IF (Mach_Control.Ca_b.Error[18] AND Sys_Control.btn.System_Rrestbtn) OR
    (CCD. CaRec.Finish.RectifyResult<>0 AND  CaCCDMark AND  Ca_AlarmTon[13].Q ) THEN
	   CaCCDMark :=FALSE;
	   Ca_AlarmTon[12].IN:=FALSE;
END_IF	

IF Mach_Control.U.DT_iMode=1 AND  rCaUse[4].Q THEN
 Par.stDT_date.Ca_sucker1_JS :=Par.stDT_date.Ca_sucker1_JS+1;
END_IF

IF( HMI_Hour>=7  AND HMI_Hour<9) OR (HMI_Hour>=19  AND HMI_Hour<21) THEN
      IF Par.stDT_date.Ca_sucker1_JS>=Par.stDT_date.Ca_sucker1Set THEN
	      Mach_Control.Ca_b.Error[43]:=TRUE;//负极送片搬运吸盘计数到达设定值
      END_IF
END_IF
IF Mach_Control.DT_b.Ca_sucker1_JSclear THEN
   Par.stDT_date.Ca_sucker1_JS:=0;
END_IF  

IF Mach_Control.U.DT_iMode=1 AND  rCaUse[5].Q THEN
 Par.stDT_date.Ca_sucker2_JS :=Par.stDT_date.Ca_sucker2_JS+1;
END_IF

IF( HMI_Hour>=7  AND HMI_Hour<9) OR (HMI_Hour>=19  AND HMI_Hour<21) THEN
      IF Par.stDT_date.Ca_sucker2_JS>=Par.stDT_date.Ca_sucker2Set THEN
	      Mach_Control.Ca_b.Error[44]:=TRUE;//负极叠台搬运吸盘计数到达设定值
      END_IF
END_IF
IF Mach_Control.DT_b.Ca_sucker2_JSclear THEN
   Par.stDT_date.Ca_sucker2_JS:=0;
END_IF  
IF Mach_Control.U.DT_iMode=1 AND  rCaUse[6].Q THEN
 Par.stDT_date.Ca_sucker3_JS :=Par.stDT_date.Ca_sucker3_JS+1;
END_IF

IF( HMI_Hour>=7  AND HMI_Hour<9) OR (HMI_Hour>=19  AND HMI_Hour<21) THEN
      IF Par.stDT_date.Ca_sucker3_JS>=Par.stDT_date.Ca_sucker3Set THEN
	      Mach_Control.Ca_b.Error[45]:=TRUE;//负极流水线搬运吸盘计数到达设定值
      END_IF
END_IF
IF Mach_Control.DT_b.Ca_sucker3_JSclear THEN
   Par.stDT_date.Ca_sucker3_JS:=0;
END_IF  
(*
IF Ca_CCDNG>=10 THEN
		Mach_Control.Ca_b.Error[12]:=TRUE;//负极NG收纳盒满料报警
END_IF

IF Mach_Control.Ca_b.Error[12] AND P2M2_sysControl.btn.System_Rrestbtn THEN
		 Mach_Control.Ca_b.Error[12]:=FALSE;
		 Ca_CCDNG:=0;
END_IF

*)
END_ACTION

ACTION Ca_Cahebelt:
Ca_TON[9].IN:=Mach_Control.Ca_b.bCa_PoleHave;
IF Ca_TON[9].Q THEN
	Mach_Control.Ca_b.bCa_PoleHave:=FALSE;//负极取流水线极片完成，
END_IF


//取料中信号复位
Ca_TON[10].IN:= NOT  arrAxisCtrl[AxiseNo.AxisName.CaCarryingUpDown1].Cmd.arrbRealPoint[1] AND Mach_Control.Ca_b.JumpPiceReady AND Mach_Control.Ca_b.Ca_MainBelting;
IF Ca_TON[10].Q THEN
	IF NOT  arrAxisCtrl[AxiseNo.AxisName.CaCarryingUpDown1].Cmd.arrbRealPoint[1] THEN		
		arrAxisCtrl[AxiseNo.AxisName.CaCarryingUpDown1].Cmd.iGoSetPos:=1;//负极送片搬运升降上升至初始高度	
	ELSE
		arrAxisCtrl[AxiseNo.AxisName.CaCarryingUpDown1].Cmd.iGoSetPos:=0;//负极送片搬运升降上升至初始高度	
	END_IF
END_IF
Ca_TON[11].IN:=arrAxisCtrl[AxiseNo.AxisName.CaCarryingUpDown1].Cmd.arrbRealPoint[1] AND Mach_Control.Ca_b.JumpPiceReady AND Mach_Control.Ca_b.Ca_MainBelting;
IF Ca_TON[11].Q  THEN
	Ca_StandbyStep2:=0;
	Mach_Control.Ca_b.Ca_BeltDone:=TRUE;//取流水线取极片完成
	Mach_Control.Ca_b.Ca_MainBelting:=FALSE;//正极搬运升降取极片中
END_IF




IF Mach_Control.U.DT_iMode=1 OR AG  THEN//在自动状态下
//负极模切分段皮带极片自动
CASE Ca_StandbyStep2  OF
0://判断取模切分板皮带机械手有无料标记
	IF NOT DP_SinStepe THEN
		IF   arrAxisCtrl[AxiseNo.AxisName.CaCarryingUpDown1].Status.Enabled  AND  arrAxisCtrl[AxiseNo.AxisName.CaCarryingLine1].Status.Enabled 
		AND  arrAxisCtrl[AxiseNo.AxisName.CaCarryingWhirling1].Status.Enabled  THEN
			IF Mach_Control.Ca_b.Ca_SegbeltFalg  THEN//负极取模切分段机械手有极片标记
				DT_SingeMode();//单步选择
				Ca_StandbyStep2:=100;
			ELSE//负极取模切分段机械手无料
				
				DT_SingeMode();//单步选择
				Ca_StandbyStep2:=10;
			END_IF
		END_IF
	END_IF
10://负极送片搬运升降轴上升至安全位，真空关闭
	IF NOT DP_SinStepe THEN
		arrCyCtrl[arrCyNo.ElectValveName.CaCarryingVacuum1]	.Cmd.bOFF:=TRUE;//负极搬运1真空关
		arrCyCtrl[arrCyNo.ElectValveName.CaCarryingVacuum1]	.Cmd.bON:=FALSE;//负极搬运1真空开
		IF arrAxisCtrl[AxiseNo.AxisName.CaCarryingUpDown1].Status.Homed AND arrAxisCtrl[AxiseNo.AxisName.CaCarryingUpDown1].Status.NoMoving AND 
			NOT arrAxisCtrl[AxiseNo.AxisName.CaCarryingUpDown1].Status.Error THEN
				IF arrAxisCtrl[AxiseNo.AxisName.CaCarryingUpDown1].Cmd.arrbRealPoint[1] THEN
					arrAxisCtrl[AxiseNo.AxisName.CaCarryingUpDown1].Cmd.iGoSetPos:=0;
					DT_SingeMode();//单步选择
					Ca_StandbyStep2:=20;
				ELSE
					arrAxisCtrl[AxiseNo.AxisName.CaCarryingUpDown1].Cmd.iGoSetPos:=1;//负极搬运升降1移动至初始高度
				END_IF
		END_IF
	END_IF
20://负极送片搬运平移至模切分段皮带取料位,负极搬运旋转1旋转至初始位
	IF NOT DP_SinStepe THEN
		IF arrAxisCtrl[AxiseNo.AxisName.CaCarryingUpDown1].Cmd.arrbRealPoint[1] AND  arrAxisCtrl[AxiseNo.AxisName.CaCarryingLine1].Status.Homed AND 
			arrAxisCtrl[AxiseNo.AxisName.CaCarryingLine1].Status.NoMoving AND NOT arrAxisCtrl[AxiseNo.AxisName.CaCarryingLine1].Status.Error THEN
			IF arrAxisCtrl[AxiseNo.AxisName.CaCarryingLine1].Cmd.arrbRealPoint[1] THEN
				arrAxisCtrl[AxiseNo.AxisName.CaCarryingLine1].Cmd.iGoSetPos:=0;
			ELSE
				arrAxisCtrl[AxiseNo.AxisName.CaCarryingLine1].Cmd.iGoSetPos:=1;//负极搬运升降1移动至初始高度
			END_IF
		END_IF
		IF arrAxisCtrl[AxiseNo.AxisName.CaCarryingUpDown1].Cmd.arrbRealPoint[1] AND  arrAxisCtrl[AxiseNo.AxisName.CaCarryingWhirling1].Status.Homed AND
			 arrAxisCtrl[AxiseNo.AxisName.CaCarryingWhirling1].Status.NoMoving AND NOT arrAxisCtrl[AxiseNo.AxisName.CaCarryingWhirling1].Status.Error THEN
			IF arrAxisCtrl[AxiseNo.AxisName.CaCarryingWhirling1].Cmd.arrbRealPoint[1] THEN
				arrAxisCtrl[AxiseNo.AxisName.CaCarryingWhirling1].Cmd.iGoSetPos:=0;
			ELSE
				arrAxisCtrl[AxiseNo.AxisName.CaCarryingWhirling1].Cmd.iGoSetPos:=1;//负极搬运旋转至初始位
			END_IF
		END_IF
		IF arrAxisCtrl[AxiseNo.AxisName.CaCarryingLine1].Cmd.arrbRealPoint[1]  AND arrAxisCtrl[AxiseNo.AxisName.CaCarryingWhirling1].Cmd.arrbRealPoint[1] THEN
			DT_SingeMode();//单步选择
			Ca_StandbyStep2:=30;
		END_IF
	END_IF

	

100://负极送片搬运升降轴上升至安全位，真空关闭
	IF NOT DP_SinStepe THEN
		IF arrAxisCtrl[AxiseNo.AxisName.CaCarryingUpDown1].Status.Homed AND arrAxisCtrl[AxiseNo.AxisName.CaCarryingUpDown1].Status.NoMoving AND 
			NOT arrAxisCtrl[AxiseNo.AxisName.CaCarryingUpDown1].Status.Error THEN
			IF arrAxisCtrl[AxiseNo.AxisName.CaCarryingUpDown1].Cmd.arrbRealPoint[1] THEN
						arrAxisCtrl[AxiseNo.AxisName.CaCarryingUpDown1].Cmd.iGoSetPos:=0;
						DT_SingeMode();//单步选择
						Ca_StandbyStep2:=110;
			ELSE
				arrAxisCtrl[AxiseNo.AxisName.CaCarryingUpDown1].Cmd.iGoSetPos:=1;//负极搬运升降1移动至初始高度
			END_IF
		END_IF
	END_IF
110://负极送片搬运平移至模切分段皮带放极片位, 负极搬运旋转1旋转至放位
	IF NOT DP_SinStepe THEN
		IF arrAxisCtrl[AxiseNo.AxisName.CaCarryingUpDown1].Cmd.arrbRealPoint[1] AND  arrAxisCtrl[AxiseNo.AxisName.CaCarryingLine1].Status.Homed AND 
			arrAxisCtrl[AxiseNo.AxisName.CaCarryingLine1].Status.NoMoving AND NOT arrAxisCtrl[AxiseNo.AxisName.CaCarryingLine1].Status.Error THEN
			IF arrAxisCtrl[AxiseNo.AxisName.CaCarryingLine1].Cmd.arrbRealPoint[2] THEN
				arrAxisCtrl[AxiseNo.AxisName.CaCarryingLine1].Cmd.iGoSetPos:=0;
			ELSE
				arrAxisCtrl[AxiseNo.AxisName.CaCarryingLine1].Cmd.iGoSetPos:=2;//负极搬运升降1移动至放极片位
			END_IF
		END_IF
		IF arrAxisCtrl[AxiseNo.AxisName.CaCarryingUpDown1].Cmd.arrbRealPoint[1] AND  arrAxisCtrl[AxiseNo.AxisName.CaCarryingWhirling1].Status.Homed AND
			 arrAxisCtrl[AxiseNo.AxisName.CaCarryingWhirling1].Status.NoMoving AND NOT arrAxisCtrl[AxiseNo.AxisName.CaCarryingWhirling1].Status.Error THEN
			IF arrAxisCtrl[AxiseNo.AxisName.CaCarryingWhirling1].Cmd.arrbRealPoint[2] THEN
				arrAxisCtrl[AxiseNo.AxisName.CaCarryingWhirling1].Cmd.iGoSetPos:=0;
			ELSE
				arrAxisCtrl[AxiseNo.AxisName.CaCarryingWhirling1].Cmd.iGoSetPos:=2;//负极搬运旋转至放极片位
			END_IF
		END_IF
		IF arrAxisCtrl[AxiseNo.AxisName.CaCarryingLine1].Cmd.arrbRealPoint[2]  AND arrAxisCtrl[AxiseNo.AxisName.CaCarryingWhirling1].Cmd.arrbRealPoint[2] THEN
			DT_SingeMode();//叠片单步选择
			Ca_StandbyStep2:=120;
		END_IF
	END_IF
120://判断负极流水线是否允许放极片  OR Mach_Control.U.EmptyRunMode
	IF NOT DP_SinStepe THEN
		IF Mach_Control.Ca_b.Ca_CacheBeltFLOK AND  Mach_Control.Ca_b.Ca_SegbeltFalg THEN
			DT_SingeMode();//单步选择
			Ca_StandbyStep2:=130;
		ELSIF NOT Mach_Control.Ca_b.Ca_SegbeltFalg THEN
			Ca_StandbyStep2:=0;
		END_IF
	END_IF
130://负极搬运升降1下降至放极片位
	IF NOT DP_SinStepe THEN
		IF arrAxisCtrl[AxiseNo.AxisName.CaCarryingLine1].Cmd.arrbRealPoint[2]  AND arrAxisCtrl[AxiseNo.AxisName.CaCarryingWhirling1].Cmd.arrbRealPoint[2] AND 
			arrAxisCtrl[AxiseNo.AxisName.CaCarryingUpDown1].Status.Homed AND arrAxisCtrl[AxiseNo.AxisName.CaCarryingUpDown1].Status.NoMoving AND 
			NOT arrAxisCtrl[AxiseNo.AxisName.CaCarryingUpDown1].Status.Error THEN
			IF arrAxisCtrl[AxiseNo.AxisName.CaCarryingUpDown1].Cmd.arrbRealPoint[3] THEN
				arrAxisCtrl[AxiseNo.AxisName.CaCarryingUpDown1].Cmd.iGoSetPos:=0;
				arrCyCtrl[arrCyNo.ElectValveName.CaCarryingVacuum1].Cmd.bOFF:=TRUE;//负极搬运1升降真空关
				arrCyCtrl[arrCyNo.ElectValveName.CaCarryingVacuum1].Cmd.bON:=FALSE;//负极搬运1升降真空关
				arrCyCtrl[arrCyNo.ElectValveName.CaCarryingVacuumBark1].Cmd.bON:=TRUE;//负极搬运1升降破真空开
				arrCyCtrl[arrCyNo.ElectValveName.CaCarryingVacuumBark1].Cmd.bOFF:=FALSE;//负极搬运1升降破真空开
				Mach_Control.Ca_b.Ca_SegbeltFalg:=FALSE;//置位负极取模切分段机械手有极片标记
				Par.stDT_date.Ca_betlCount.0:=TRUE;//置位负极片流水线放片位有片
				Par.stDT_date.Ca_MQ_Slice[1]:=Par.stDT_date.Ca_MQ_Slice[0];
				DT_SingeMode();//单步选择
				Ca_StandbyStep2:=140;
			ELSE
				arrAxisCtrl[AxiseNo.AxisName.CaCarryingUpDown1].Cmd.iGoSetPos:=3;//负极搬运升降1移动至放极片高度
			END_IF
		ELSE
			IF arrAxisCtrl[AxiseNo.AxisName.CaCarryingLine1].Cmd.arrbRealPoint[2] THEN
				arrAxisCtrl[AxiseNo.AxisName.CaCarryingLine1].Cmd.iGoSetPos:=0;
			ELSE
				arrAxisCtrl[AxiseNo.AxisName.CaCarryingLine1].Cmd.iGoSetPos:=2;//负极搬运升降1移动至放极片位
			END_IF	
			IF arrAxisCtrl[AxiseNo.AxisName.CaCarryingWhirling1].Cmd.arrbRealPoint[2] THEN
				arrAxisCtrl[AxiseNo.AxisName.CaCarryingWhirling1].Cmd.iGoSetPos:=0;
			ELSE
				arrAxisCtrl[AxiseNo.AxisName.CaCarryingWhirling1].Cmd.iGoSetPos:=2;//负极搬运旋转至放极片位
			END_IF			
		END_IF
	END_IF
140://负极送片搬运升降轴上升至安全位，真空关闭
	IF NOT DP_SinStepe THEN
		IF arrAxisCtrl[AxiseNo.AxisName.CaCarryingUpDown1].Status.Homed AND arrAxisCtrl[AxiseNo.AxisName.CaCarryingUpDown1].Status.NoMoving AND 
			NOT arrAxisCtrl[AxiseNo.AxisName.CaCarryingUpDown1].Status.Error THEN
			IF arrAxisCtrl[AxiseNo.AxisName.CaCarryingUpDown1].Cmd.arrbRealPoint[1] THEN
				arrAxisCtrl[AxiseNo.AxisName.CaCarryingUpDown1].Cmd.iGoSetPos:=0;
				DT_SingeMode();//单步选择
				Ca_StandbyStep2:=0;
			ELSE
				arrAxisCtrl[AxiseNo.AxisName.CaCarryingUpDown1].Cmd.iGoSetPos:=1;//负极搬运升降1移动至初始高度
			END_IF
		END_IF
	END_IF				
END_CASE	
END_IF


//负极缓存流水线缓存极片自动	
CASE Ca_StandbyStep4 OF
0://判断是否可以补极片,负极搬运升降1轴在安全位，负极搬运各项降2轴在安全位，负极流水线放极片端有极片，负极片流水线取级片端没极片 
	IF NOT Par.stDT_date.Ca_betlCount.5 AND Par.stDT_date.Ca_betlCount.0 AND  Mach_Control.Ca_b.Ca_betlMoveOK  THEN
		IF NOT Mach_Control.se.Offloadingsensor THEN
				Par.stDT_date.Ca_betlCount.4:=FALSE;
		END_IF
		Ca_StandbyStep4:=10;
	ELSIF	Ca_StandbyStep2=120 AND NOT Par.stDT_date.Ca_betlCount.5 AND Par.stDT_date.Ca_betlCount.0  AND  NOT  arrAxisCtrl[AxiseNo.AxisName.CaCarryingUpDown1].Cmd.arrbRealPoint[1] THEN
               // ( arrAxisCtrl[AxiseNo.AxisName.CaCarryingUpDown1].Status.fSetPos > arrAxisPar[AxiseNo.AxisName.CaCarryingUpDown1].arrTargetPoint[1]+0.5 OR
                //  arrAxisCtrl[AxiseNo.AxisName.CaCarryingUpDown1].Status.fSetPos < arrAxisPar[AxiseNo.AxisName.CaCarryingUpDown1].arrTargetPoint[1]-0.5)THEN
		         Mach_Control.Ca_b.Error[41]:=TRUE;//负极缓存皮带准备运动时，负极升降1不在安全位报警	
	END_IF
10://负极流水线皮带向前移动固定距离
	arrAxisCtrl[AxiseNo.AxisName.CaBelt].Cmd.bDynamitcsParSel:=1;	
	arrAxisPar[AxiseNo.AxisName.CaBelt].fTagatTime:=Par.stDT_date.BeltPoistTime;
	arrAxisCtrl[AxiseNo.AxisName.CaBelt].Cmd.fPosition_of_Rel:=Par.stDT_date.BeltPoistSet;
	arrAxisCtrl[AxiseNo.AxisName.CaBelt].Cmd.bMoveRel:=TRUE;	
	Ca_StandbyStep4:=20;
20:
	IF NOT arrAxisCtrl[AxiseNo.AxisName.CaBelt].Cmd.bMoveRel THEN
		Par.stDT_date.Ca_betlCount:=SHL(Par.stDT_date.Ca_betlCount,1);//极片向前移一位
		Ca_StandbyStep4:=31;
	END_IF

31:	
	Par.stDT_date.Ca_MQ_Slice[6]:=Par.stDT_date.Ca_MQ_Slice[5];
	Ca_StandbyStep4:=32;

32:
	Par.stDT_date.Ca_MQ_Slice[5]:=Par.stDT_date.Ca_MQ_Slice[4];
	Ca_StandbyStep4:=33;

33:
	Par.stDT_date.Ca_MQ_Slice[4]:=Par.stDT_date.Ca_MQ_Slice[3];
	Ca_StandbyStep4:=34;

34:	
	Par.stDT_date.Ca_MQ_Slice[3]:=Par.stDT_date.Ca_MQ_Slice[2];
	Ca_StandbyStep4:=35;

35:
	Par.stDT_date.Ca_MQ_Slice[2]:=Par.stDT_date.Ca_MQ_Slice[1];
	Ca_StandbyStep4:=36;

36://复位负极片流水线放片位有片
	MEMSET(ADR(Par.stDT_date.Ca_MQ_Slice[1]),0,SIZEOF(Par.stDT_date.Ca_MQ_Slice[1]));
	Par.stDT_date.Ca_betlCount.0:=FALSE;
	Ca_StandbyStep4:=0;
END_CASE


CASE Ca_StandbyStep2  OF
30://判断模切分段皮带是否允许取极片 OR Mach_Control.U.EmptyRunMode 
	IF NOT DP_SinStepe THEN
		IF Mach_Control.Ca_b.Ca_MainBeltOK THEN
			Mach_Control.Ca_b.Ca_MainBelting:=TRUE;//负极模切分段皮带取极片中
			arrCyCtrl[arrCyNo.ElectValveName.CaCarryingVacuum1]	.Cmd.bON:=TRUE;//负极搬运1真空打开
			arrCyCtrl[arrCyNo.ElectValveName.CaCarryingVacuum1]	.Cmd.bOFF:=FALSE;//负极搬运1真空关闭
			DT_SingeMode();//单步选择
			Ca_StandbyStep2:=35;
		//ELSE
		//	Ca_StandbyStep2:=0;
		END_IF
	END_IF
35://负极搬动升降1下降取极片
	IF NOT DP_SinStepe THEN
		IF arrAxisCtrl[AxiseNo.AxisName.CaCarryingLine1].Cmd.arrbRealPoint[1]  AND arrAxisCtrl[AxiseNo.AxisName.CaCarryingWhirling1].Cmd.arrbRealPoint[1] AND 
			arrAxisCtrl[AxiseNo.AxisName.CaCarryingUpDown1].Status.Homed AND  NOT arrAxisCtrl[AxiseNo.AxisName.CaCarryingUpDown1].Status.Error THEN
			IF arrAxisCtrl[AxiseNo.AxisName.CaCarryingUpDown1].Cmd.arrbRealPoint[2] OR arrAxisCtrl[AxiseNo.AxisName.CaCarryingUpDown1].Status.Moving THEN
				arrAxisCtrl[AxiseNo.AxisName.CaCarryingUpDown1].Cmd.iGoSetPos:=0;
				DT_SingeMode();//单步选择
				Ca_TON[6].IN:=FALSE;
				Ca_StandbyStep2:=40;
			ELSE
				arrAxisCtrl[AxiseNo.AxisName.CaCarryingUpDown1].Cmd.iGoSetPos:=2;//负极搬运升降1移动至初始高度
			END_IF					
		END_IF
	END_IF
40://负极搬动升降1下降取极片
	IF arrAxisCtrl[AxiseNo.AxisName.CaCarryingLine1].Cmd.arrbRealPoint[1]  AND arrAxisCtrl[AxiseNo.AxisName.CaCarryingWhirling1].Cmd.arrbRealPoint[1] AND 
	arrAxisCtrl[AxiseNo.AxisName.CaCarryingUpDown1].Status.Homed AND arrAxisCtrl[AxiseNo.AxisName.CaCarryingUpDown1].Status.NoMoving AND 
	NOT arrAxisCtrl[AxiseNo.AxisName.CaCarryingUpDown1].Status.Error THEN
		IF arrAxisCtrl[AxiseNo.AxisName.CaCarryingUpDown1].Cmd.arrbRealPoint[2] THEN			
			IF NOT Ca_TON[6].Q THEN
				Ca_TON[6].IN:=TRUE;
			ELSE
				//Mach_Control.Ca_b.bCa_PoleHave:=TRUE;//负极取流水线极片完成，复位取片位置极片有无信号
				arrAxisCtrl[AxiseNo.AxisName.CaCarryingUpDown1].Cmd.iGoSetPos:=0;
				//arrCyCtrl[arrCyNo.ElectValveName.CaMQBeltVacuum].Cmd.bOFF:=TRUE;//负极模切分段皮带真空关闭
				//arrCyCtrl[arrCyNo.ElectValveName.CaMQBeltVacuum].Cmd.bON:=FALSE;//负极模切分段皮带真空关闭
				//arrCyCtrl[arrCyNo.ElectValveName.CaMQBeltVacuumBark].Cmd.bON:=TRUE;//负极模切分段皮带破真空打开
				Mach_Control.Ca_b.Ca_SegbeltFalg:=TRUE;//置位负极取模切分段机械手有极片标记
				Par.stDT_date.Ca_MQ_Slice[0]:=Par.stDT_date.CaMQ_MES;//转移皮带上的数据
				DT_SingeMode();//单步选择
				Ca_TON[6].IN:=FALSE;
				Ca_StandbyStep2:=50;								
			END_IF								
		ELSE
			arrAxisCtrl[AxiseNo.AxisName.CaCarryingUpDown1].Cmd.iGoSetPos:=2;//负极搬运升降1移动至初始高度
		END_IF					
	END_IF

50://
	//20240414 wcz
    IF   arrAxisCtrl[AxiseNo.AxisName.CaCarryingUpDown1].Status.fActPos<=(arrAxisPar[AxiseNo.AxisName.CaCarryingUpDown1].arrTargetPoint[2]-3) AND
		 arrAxisCtrl[AxiseNo.AxisName.CaCarryingUpDown1].Status.Moving THEN
			Mach_Control.Ca_b.Ca_MainBelting:=FALSE;//负极模切分段皮带取极片中
			Mach_Control.Ca_b.Ca_BeltDone:=TRUE;//负极取主流水线极片完成		 
			Mach_Control.Ca_b.bCa_PoleHave:=TRUE;//负极取流水线极片完成，复位取片位置极片有无信号
	END_IF

	IF arrAxisCtrl[AxiseNo.AxisName.CaCarryingUpDown1].Status.Homed AND arrAxisCtrl[AxiseNo.AxisName.CaCarryingUpDown1].Status.NoMoving AND 
	NOT arrAxisCtrl[AxiseNo.AxisName.CaCarryingUpDown1].Status.Error THEN
		IF arrAxisCtrl[AxiseNo.AxisName.CaCarryingUpDown1].Cmd.arrbRealPoint[1] THEN
			arrAxisCtrl[AxiseNo.AxisName.CaCarryingUpDown1].Cmd.iGoSetPos:=0;
			Mach_Control.Ca_b.Ca_MainBelting:=FALSE;//负极模切分段皮带取极片中
			Mach_Control.Ca_b.Ca_BeltDone:=TRUE;//负极取主流水线极片完成
			DT_SingeMode();//单步选择
			Ca_StandbyStep2:=0;
		ELSE
			arrAxisCtrl[AxiseNo.AxisName.CaCarryingUpDown1].Cmd.iGoSetPos:=1;//负极搬运升降1移动至初始高度
		END_IF
	END_IF
END_CASE
END_ACTION

ACTION Ca_Cam:
Ca_Cam_ton[1](PT:=T#100MS);
Ca_Cam_ton[2](PT:=T#100MS);
Ca_Cam_ton[3](PT:=T#100MS);
Ca_Cam_ton[4](PT:=T#100MS);
Ca_Cam_ton[5](PT:=T#100MS);
(***********************************负极凸轮表创建************************************************)
(*
      fbCaCrectCamCarryingLine1              :FB_CrectCamMove ;
      fbCaCrectCamCarryingUpDown1       :FB_CrectCamUpDown ;
      fbCaCrectCamCarryingLine2             :FB_CrectCamMove ;
      fbCaCrectCamCarryingUpDown2       :FB_CrectCamUpDown ;
      fbCaCrectCamDTCarryingLine            :FB_CrectCamMove ;
      fbCaCrectCamDTCarryingUpDown     :FB_CrectCamUpDown ;
*)
//负极取流水线搬运平移凸轮创建
fbCaCrectCamCarryingLine1(
	bCreatTable:=                fbCaCrectCamCarryingLine1.bCreatTable , 
	Reset:=                          stSysState.bReset  ,  
	iTable:=                       TableNo.M_CaCarryingLine1  , 
	fMoveLength:=             390 , 
	fMasterKeyPos:=          224 , 
	
	axisMaster:=                 arrAxis[AxiseNo.VirAxisName.CaCarryingVirGM] ,  
    axisSlave:=                    arrAxis[AxiseNo.AxisName.CaCarryingLine1] ,  
	bCreatTableDone=> , 
	bCreatTableError=> , 
	bError=> );

fbCaCrectCamCarryingLine1.bCreatTableDone;
fbCaCrectCamCarryingLine1.bCreatTableError;
fbCaCrectCamCarryingLine1.bError;

//负极取流水线搬运放片升降凸轮创建
fbCaCrectCamCarryingUpDown1(
	bCreatTable:=                         fbCaCrectCamCarryingUpDown1.bCreatTable , 
	Reset:=                                  stSysState.bReset  ,  
	iTable:=                                   TableNo.M_CaCarryingUpDown1   , 
	fMoveLength:=                        18   , //升降轴放片或取片位
	fSaveLength:=                          3, //升降轴安全位
	fInitLength:=						      13,//升降轴耦合初始位
	fMasterKeyPos1:= , //208
	fMasterKeyPos2:= , //256
	fMasterKeyPos3:= , //328

    axisMaster:=                        arrAxis[AxiseNo.VirAxisName.CaCarryingVirGM] ,   
	axisSlave:=                           arrAxis[AxiseNo.AxisName.CaCarryingUpDown1] ,  

	bCreatTableDone=> , 
	bCreatTableError=> , 
	bError=> );
fbCaCrectCamCarryingUpDown1.bCreatTableDone;
fbCaCrectCamCarryingUpDown1.bCreatTableError;
fbCaCrectCamCarryingUpDown1.bError;

//负极取流水线搬运取片升降凸轮创建
fbCaCrectCamCarryingUpDown1_1(
	bCreatTable:=                         fbCaCrectCamCarryingUpDown1_1.bCreatTable , 
	Reset:=                                  stSysState.bReset  ,  
	iTable:=                                   TableNo.M_CaCarryingUpDown1_1   , 
	fMoveLength:=                        18   , //升降轴放片或取片位
	fSaveLength:=                          3, //升降轴安全位
	fInitLength:=						      13,//升降轴耦合初始位
	fMasterKeyPos1:= , //208
	fMasterKeyPos2:= , //256
	fMasterKeyPos3:= , //328

    axisMaster:=                        arrAxis[AxiseNo.VirAxisName.CaCarryingVirGM] ,   
	axisSlave:=                           arrAxis[AxiseNo.AxisName.CaCarryingUpDown1] ,  

	bCreatTableDone=> , 
	bCreatTableError=> , 
	bError=> );
fbCaCrectCamCarryingUpDown1_1.bCreatTableDone;
fbCaCrectCamCarryingUpDown1_1.bCreatTableError;
fbCaCrectCamCarryingUpDown1_1.bError;

//负极取流水线旋转凸轮创建 
fbCaCrectCamCarryingWhirling(
	bCreatTable:=                fbCaCrectCamCarryingWhirling.bCreatTable , 
	Reset:=                          stSysState.bReset  ,  
	iTable:=                       TableNo.M_CaCarryingWhirling1  , 
	fMoveLength:=             390 , 
	fMasterKeyPos:=          170 , //224
	
	axisMaster:=                 arrAxis[AxiseNo.VirAxisName.CaCarryingVirGM] ,  
    axisSlave:=                    arrAxis[AxiseNo.AxisName.CaCarryingWhirling1] ,  
	bCreatTableDone=> , 
	bCreatTableError=> , 
	bError=> );

fbCaCrectCamCarryingWhirling.bCreatTableDone;
fbCaCrectCamCarryingWhirling.bCreatTableError;
fbCaCrectCamCarryingWhirling.bError;




//负极送纠偏平台搬运平移凸轮创建
fbCaCrectCamCarryingLine2.fMoveLength:=ABS(arrAxisPar[AxiseNo.AxisName.CaCarryingLine2].arrTargetPoint[1]-arrAxisPar[AxiseNo.AxisName.CaCarryingLine2].arrTargetPoint[2]);
fbCaCrectCamCarryingLine2(
	bCreatTable:=                fbCaCrectCamCarryingLine2.bCreatTable , 
	Reset:=                          stSysState.bReset  ,  
	iTable:=                       TableNo.M_CaCarryingLine2  , 
	fMoveLength:=             , 
	fMasterKeyPos:=          250 , //
	
	axisMaster:=                 arrAxis[AxiseNo.VirAxisName.VirMain] ,  
    axisSlave:=                    arrAxis[AxiseNo.AxisName.CaCarryingLine2] ,  
	bCreatTableDone=> , 
	bCreatTableError=> , 
	bError=> );

fbCaCrectCamCarryingLine2.bCreatTableDone;
fbCaCrectCamCarryingLine2.bCreatTableError;
fbCaCrectCamCarryingLine2.bError;


(**********20240528SJ***************)
arrAxisPar[AxiseNo.AxisName.CaCarryingUpDown2].arrTargetPoint[10]:=10; //等待高度  参数可调
arrAxisPar[AxiseNo.AxisName.CaCarryingUpDown2].arrTargetPoint[11]:=25; //安全高度  参数可调
arrAxisPar[AxiseNo.AxisName.CaCarryingUpDown2].arrTargetPoint[4]:=arrAxisPar[AxiseNo.AxisName.CaCarryingUpDown2].arrTargetPoint[3]-arrAxisPar[AxiseNo.AxisName.CaCarryingUpDown2].arrTargetPoint[10];  //等待位置
//arrAxisPar[AxiseNo.AxisName.AnCarryingUpDown].arrTargetPoint[1]:=arrAxisPar[AxiseNo.AxisName.AnCarryingUpDown].arrTargetPoint[3]-arrAxisPar[AxiseNo.AxisName.AnCarryingUpDown].arrTargetPoint[11];  //安全位置

//负极送纠偏平台搬运升降取片凸轮创建 20240509 CF
fbCaCrectCamCarryingUpDown2(  //取片
	bCreatTable:=                         fbCaCrectCamCarryingUpDown2.bCreatTable , 
	Reset:=                                  stSysState.bReset  ,  
	iTable:=                                   TableNo.M_CaCarryingUpDown2   , 
	fMoveLength:=4, //取片高度
	fSaveLength:=arrAxisPar[AxiseNo.AxisName.CaCarryingUpDown2].arrTargetPoint[10] - arrAxisPar[AxiseNo.AxisName.CaCarryingUpDown2].arrTargetPoint[11],//安全高度
	//fInitLength:=arrAxisPar[AxiseNo.AxisName.CaCarryingUpDown2].arrTargetPoint[4],//升降轴耦合初始位
	fMasterKeyPos1:=110 , //
	fMasterKeyPos2:=250 , //144
	//fMasterKeyPos3:=240 , //198
	//fMasterKeyPos4:=310 , //324
	
    axisMaster:=                        arrAxis[AxiseNo.VirAxisName.VirMain] ,   
	axisSlave:=                           arrAxis[AxiseNo.AxisName.CaCarryingUpDown2] ,  

	bCreatTableDone=> , 
	bCreatTableError=> , 
	bError=> );
fbCaCrectCamCarryingUpDown2.bCreatTableDone;
fbCaCrectCamCarryingUpDown2.bCreatTableError;
fbCaCrectCamCarryingUpDown2.bError;


//负极送纠偏平台搬运升降放极片凸轮创建-
fbCaCrectCamCarryingUpDown2_1(   //--------放片
	bCreatTable:=                         fbCaCrectCamCarryingUpDown2_1.bCreatTable , 
	Reset:=                                  stSysState.bReset  ,  
	iTable:=                                   TableNo.M_CaCarryingUpDown2_1   , 
	fMoveLength:= arrAxisPar[AxiseNo.AxisName.CaCarryingUpDown2].arrTargetPoint[10]       ,//放片高度
	fSaveLength:=arrAxisPar[AxiseNo.AxisName.CaCarryingUpDown2].arrTargetPoint[10] - arrAxisPar[AxiseNo.AxisName.CaCarryingUpDown2].arrTargetPoint[11]  , //安全高度
	//fInitLength:=arrAxisPar[AxiseNo.AxisName.CaCarryingUpDown2].arrTargetPoint[4],//升降轴耦合初始位
	fMasterKeyPos1:=110 , //125
	fMasterKeyPos2:=250 , //
	fMasterKeyPos3:=260 , //
	fMasterKeyPos4:=320 , //
	fMasterKeyPos5:=359 , //
	//fMasterKeyPos6:=250 , //
	fSlaveVelo:=0.25 , //
	
    axisMaster:=                        arrAxis[AxiseNo.VirAxisName.VirMain] ,   
	axisSlave:=                           arrAxis[AxiseNo.AxisName.CaCarryingUpDown2] ,  

	bCreatTableDone=> , 
	bCreatTableError=> , 
	bError=> );
fbCaCrectCamCarryingUpDown2_1.bCreatTableDone;
fbCaCrectCamCarryingUpDown2_1.bCreatTableError;
fbCaCrectCamCarryingUpDown2_1.bError;

//负极送纠偏平台搬运升降放极片凸轮创建-
fbCaCrectCamCarryingUpDown2_3(   //--------放片
	bCreatTable:=                         fbCaCrectCamCarryingUpDown2_3.bCreatTable , 
	Reset:=                                   stSysState.bReset  ,  
	iTable:=                                  TableNo.M_CaCarryingUpDown2_3   , 
	//fMoveLength:= arrAxisPar[AxiseNo.AxisName.CaCarryingUpDown2].arrTargetPoint[10]       ,//放片高度
	fSaveLength:=arrAxisPar[AxiseNo.AxisName.CaCarryingUpDown2].arrTargetPoint[10] - arrAxisPar[AxiseNo.AxisName.CaCarryingUpDown2].arrTargetPoint[11]  , //安全高度
	//fInitLength:=arrAxisPar[AxiseNo.AxisName.CaCarryingUpDown2].arrTargetPoint[4],//升降轴耦合初始位
	fMasterKeyPos1:=110 , //130
	fMasterKeyPos2:=250 , //
	//fMasterKeyPos3:=260 , //
	//fMasterKeyPos4:=320 , //
	//fMasterKeyPos5:=359 , //
	//fMasterKeyPos6:=250 , //
	//fSlaveVelo:=0.25 , //
	
    axisMaster:=                        arrAxis[AxiseNo.VirAxisName.VirMain] ,   
	axisSlave:=                           arrAxis[AxiseNo.AxisName.CaCarryingUpDown2] ,  

	bCreatTableDone=> , 
	bCreatTableError=> , 
	bError=> );
fbCaCrectCamCarryingUpDown2_3.bCreatTableDone;
fbCaCrectCamCarryingUpDown2_3.bCreatTableError;
fbCaCrectCamCarryingUpDown2_3.bError;




//负极叠片搬运平移凸轮创建
fbCaCrectCamDTCarryingLine.fMoveLength:=ABS(arrAxisPar[AxiseNo.AxisName.CaDTCarryingLine].arrTargetPoint[1]- arrAxisPar[AxiseNo.AxisName.CaDTCarryingLine].arrTargetPoint[2]);
fbCaCrectCamDTCarryingLine(
	bCreatTable:=                fbCaCrectCamDTCarryingLine.bCreatTable , 
	Reset:=                          stSysState.bReset  ,  
	iTable:=                        TableNo.M_CaDTCarryingLine  , 
	fMoveLength:=              , 
	fMasterKeyPos:=          250 , //
	
	axisMaster:=                 arrAxis[AxiseNo.VirAxisName.VirMain] ,  
    axisSlave:=                    arrAxis[AxiseNo.AxisName.CaDTCarryingLine] ,  
	bCreatTableDone=> , 
	bCreatTableError=> , 
	bError=> );

fbCaCrectCamDTCarryingLine.bCreatTableDone;
fbCaCrectCamDTCarryingLine.bCreatTableError;
fbCaCrectCamDTCarryingLine.bError;



(**********20240528SJ***************)
arrAxisPar[AxiseNo.AxisName.CaDTCarryingUpDown].arrTargetPoint[10]:=6; //等待高度  参数可调
arrAxisPar[AxiseNo.AxisName.CaDTCarryingUpDown].arrTargetPoint[11]:=18; //抬升高度  参数可调
arrAxisPar[AxiseNo.AxisName.CaDTCarryingUpDown].arrTargetPoint[4]:=arrAxisPar[AxiseNo.AxisName.CaDTCarryingUpDown].arrTargetPoint[3]-arrAxisPar[AxiseNo.AxisName.CaDTCarryingUpDown].arrTargetPoint[10];  //等待位置    以放片位为基准
//arrAxisPar[AxiseNo.AxisName.AnDTCarryingUpDown].arrTargetPoint[1]:=arrAxisPar[AxiseNo.AxisName.AnDTCarryingUpDown].arrTargetPoint[3]-arrAxisPar[AxiseNo.AxisName.AnDTCarryingUpDown].arrTargetPoint[11];  //安全位置

//负极叠片搬运升降取片凸轮创建
fbCaCrectCamDTCarryingUpDown(//取片
	bCreatTable:=                         fbCaCrectCamDTCarryingUpDown.bCreatTable , 
	Reset:=                                  stSysState.bReset  ,  
	iTable:=                                   TableNo.M_CaDTCarryingUpDown   , 
	fMoveLength:=arrAxisPar[AxiseNo.AxisName.CaDTCarryingUpDown].arrTargetPoint[10]-(arrAxisPar[AxiseNo.AxisName.CaDTCarryingUpDown].arrTargetPoint[3]-arrAxisPar[AxiseNo.AxisName.CaDTCarryingUpDown].arrTargetPoint[2])               ,//取片高度
	fSaveLength:=arrAxisPar[AxiseNo.AxisName.CaDTCarryingUpDown].arrTargetPoint[10]-arrAxisPar[AxiseNo.AxisName.CaDTCarryingUpDown].arrTargetPoint[11]              , //安全位
	//fInitLength:=arrAxisPar[AxiseNo.AxisName.CaDTCarryingUpDown].arrTargetPoint[4],//升降轴耦合初始位
	fMasterKeyPos1:=125 , //
	fMasterKeyPos2:=250 , //
	fMasterKeyPos3:=260 , //
	fMasterKeyPos4:= 320, //
	fMasterKeyPos5:=359 , //
	fMasterKeyPos6:= , //
	fSlaveVelo:=0.25 , //
	
    axisMaster:=                        arrAxis[AxiseNo.VirAxisName.VirMain] ,   
	axisSlave:=                           arrAxis[AxiseNo.AxisName.CaDTCarryingUpDown] ,  

	bCreatTableDone=> , 
	bCreatTableError=> , 
	bError=> );
fbCaCrectCamDTCarryingUpDown.bCreatTableDone;
fbCaCrectCamDTCarryingUpDown.bCreatTableError;
fbCaCrectCamDTCarryingUpDown.bError;


//负极叠片搬运升降放片凸轮创建
IF  DP_Step0>3000 AND DP_Step0<=3080 THEN
     fbCaCrectCamDTCarryingUpDown1.iTableSel:=2;
ELSE	 
	 fbCaCrectCamDTCarryingUpDown1.iTableSel:=1;
END_IF		 

fbCaCrectCamDTCarryingUpDown1(//放片
	bCreatTable:=                         fbCaCrectCamDTCarryingUpDown1.bCreatTable , 
	Reset:=                                   stSysState.bReset  ,  
	iTable:=                                   TableNo.M_CaDTCarryingUpDown1   , 
	bCamIn:=  fbCaCamInDTCarryingUpDown.bCamInExecute AND  fbCaCamInDTCarryingUpDown.iTableSel=2    , 
	fMoveLength:=arrAxisPar[AxiseNo.AxisName.CaDTCarryingUpDown].arrTargetPoint[10] , //取片高度
	fSaveLength:=arrAxisPar[AxiseNo.AxisName.CaDTCarryingUpDown].arrTargetPoint[10]-arrAxisPar[AxiseNo.AxisName.CaDTCarryingUpDown].arrTargetPoint[11]  , //安全高度
	//fInitLength:=arrAxisPar[AxiseNo.AxisName.CaDTCarryingUpDown].arrTargetPoint[4] ,//升降轴耦合初始位
	fMasterKeyPos1:=120 , //208
	fMasterKeyPos2:=250 , //256
	fMasterKeyPos3:=260 , //256
	fMasterKeyPos4:=342 , //328
	fMasterKeyPos5:=359 , //328
	fSlaveVelo:=0.25 , //
    axisMaster:=                        arrAxis[AxiseNo.VirAxisName.VirMain] ,   
	axisSlave:=                           arrAxis[AxiseNo.AxisName.CaDTCarryingUpDown] ,  

	bCreatTableDone=> , 
	bCreatTableError=> , 
	bError=> );
fbCaCrectCamDTCarryingUpDown1.bCreatTableDone;
fbCaCrectCamDTCarryingUpDown1.bCreatTableError;
fbCaCrectCamDTCarryingUpDown1.bError;


//正极叠片搬运升降避让凸轮创建
fbCaCrectCamDTCarryingUpDown3(//放片
	bCreatTable:=fbCaCrectCamDTCarryingUpDown3.bCreatTable, 
	Reset:=stSysState.bReset  , 
	iTable:=TableNo.M_CaDTCarryingUpDown3 , 
	//fMoveLength:=arrAxisPar[AxiseNo.AxisName.AnDTCarryingUpDown].arrTargetPoint[10] ,//放片高度 
	fSaveLength:=arrAxisPar[AxiseNo.AxisName.CaDTCarryingUpDown].arrTargetPoint[10]-arrAxisPar[AxiseNo.AxisName.CaDTCarryingUpDown].arrTargetPoint[11]  , //安全高度
	//fInitLength:=arrAxisPar[AxiseNo.AxisName.AnDTCarryingUpDown].arrTargetPoint[4],//升降轴耦合初始位
	fMasterKeyPos1:=130 , //208
	fMasterKeyPos2:=260 , //256
	//fMasterKeyPos3:=260 , //256
	//fMasterKeyPos4:=342 , //328
//	fMasterKeyPos5:=359 , //328
//	fSlaveVelo:=0.25 , //
	axisSlave:=arrAxis[AxiseNo.AxisName.CaDTCarryingUpDown]  , 
	axisMaster:=arrAxis[AxiseNo.VirAxisName.VirMain]  , 
	bCreatTableDone=> , 
	bCreatTableError=> , 
	bError=> );
	
fbCaCrectCamDTCarryingUpDown3.bCreatTableDone;
fbCaCrectCamDTCarryingUpDown3.bCreatTableError;
fbCaCrectCamDTCarryingUpDown3.bError;











tCaCreate_TON(IN:= , PT:=T#0.5S , Q=> , ET=> );
IF Mach_Control.U.DT_iMode=3 OR Mach_Control.U.DT_iMode=0 THEN//在手动状态下
				//在触摸屏上生成凸轮
				//rCaCreate_TRIG(CLK:=Mach_Control.Ca_b.CreateCamStart , Q=> );	
				rCaCreate_TRIG(CLK:=(Mach_Control.Ca_b.CreateCamStart 
                                    AND	NOT arrAxisCtrl[AxiseNo.AxisName.CaCarryingLine2].Status.Coupled
									AND	NOT arrAxisCtrl[AxiseNo.AxisName.CaCarryingUpDown2].Status.Coupled
									AND	NOT arrAxisCtrl[AxiseNo.AxisName.CaDTCarryingLine].Status.Coupled
									AND	NOT arrAxisCtrl[AxiseNo.AxisName.CaDTCarryingUpDown].Status.Coupled), Q=> );				
				IF rCaCreate_TRIG.Q THEN
					tCaCreate_TON.IN:=FALSE;
					CaCrectCamStep0:=10;
					Mach_Control.Ca_b.Error[0]:=FALSE;
				END_IF
END_IF
				//负极取料凸轮自动创建
				CASE CaCrectCamStep0 OF
						10:
								IF NOT tCaCreate_TON.Q THEN
										//fbCaCrectCamCarryingLine1.bCreatTable :=TRUE;//负极取流水线平移凸轮创建
										//fbCaCrectCamCarryingUpDown1.bCreatTable:=TRUE;//负极取流水线放片升降凸轮创建
										//fbCaCrectCamCarryingUpDown1_1.bCreatTable:=TRUE;//负极取流水线取片升降凸轮创建
										//fbCaCrectCamCarryingWhirling.bCreatTable:=TRUE;//负极取流水线旋转凸轮创建
										 fbCaCrectCamCarryingLine2.bCreatTable :=FALSE;//负极送片搬运平移凸轮创建
										 fbCaCrectCamCarryingUpDown2.bCreatTable:=FALSE;//负极送片搬运升降取片凸轮创建
										 fbCaCrectCamCarryingUpDown2_1.bCreatTable:=FALSE;//负极送片搬运升降放片凸轮创建
										 fbCaCrectCamCarryingUpDown2_3.bCreatTable:=FALSE;//负极送片搬运升降放片凸轮创建
										 fbCaCrectCamDTCarryingLine.bCreatTable :=FALSE;//负极叠片搬运平移凸轮创建
										 fbCaCrectCamDTCarryingUpDown.bCreatTable:=FALSE;//负极叠片搬运升降取片凸轮创建
										 fbCaCrectCamDTCarryingUpDown1.bCreatTable:=FALSE;//负极叠片搬运升降放片凸轮创建
										  fbCaCrectCamDTCarryingUpDown3.bCreatTable:=FALSE;//负极叠片搬运升降放片凸轮创建
										 Mach_Control.Ca_b.CreateCamDone:=FALSE;
										 tCaCreate_TON.IN:=TRUE;					
								ELSE
											tCaCreate_TON.IN:=FALSE;	
											CaCrectCamStep0:=11;
								END_IF
								
						11:	
								IF  NOT Ca_Cam_ton[1].Q THEN
									arrAxisCtrl[AxiseNo.AxisName.CaCarryingLine2].Cmd.bStop:=TRUE;
									arrAxisCtrl[AxiseNo.AxisName.CaCarryingUpDown2].Cmd.bStop:=TRUE;
									arrAxisCtrl[AxiseNo.AxisName.CaDTCarryingLine].Cmd.bStop:=TRUE;
									arrAxisCtrl[AxiseNo.AxisName.CaDTCarryingUpDown].Cmd.bStop:=TRUE;
									Ca_Cam_ton[1].IN:=TRUE;
								ELSE
									Ca_Cam_ton[1].IN:=FALSE;
									CaCrectCamStep0:=12;
									arrAxisCtrl[AxiseNo.AxisName.CaCarryingLine2].Cmd.bStop:=FALSE;
									arrAxisCtrl[AxiseNo.AxisName.CaCarryingUpDown2].Cmd.bStop:=FALSE;
									arrAxisCtrl[AxiseNo.AxisName.CaDTCarryingLine].Cmd.bStop:=FALSE;
									arrAxisCtrl[AxiseNo.AxisName.CaDTCarryingUpDown].Cmd.bStop:=FALSE;
								END_IF
								
						12:
								IF  NOT Ca_Cam_ton[2].Q THEN
									arrAxisCtrl[AxiseNo.AxisName.CaCarryingLine2].Cmd.bReset:=TRUE;	
									arrAxisCtrl[AxiseNo.AxisName.CaCarryingUpDown2].Cmd.bReset:=TRUE;
									arrAxisCtrl[AxiseNo.AxisName.CaDTCarryingLine].Cmd.bReset:=TRUE;
									arrAxisCtrl[AxiseNo.AxisName.CaDTCarryingUpDown].Cmd.bReset:=TRUE;
									Ca_Cam_ton[2].IN:=TRUE;
								 ELSE
									 Ca_Cam_ton[2].IN:=FALSE;
									 CaCrectCamStep0:=13;
									arrAxisCtrl[AxiseNo.AxisName.CaCarryingLine2].Cmd.bReset:=FALSE;	
									arrAxisCtrl[AxiseNo.AxisName.CaCarryingUpDown2].Cmd.bReset:=FALSE;
									arrAxisCtrl[AxiseNo.AxisName.CaDTCarryingLine].Cmd.bReset:=FALSE;
									arrAxisCtrl[AxiseNo.AxisName.CaDTCarryingUpDown].Cmd.bReset:=FALSE;
								 END_IF
							

						13:
							arrAxisCtrl[AxiseNo.AxisName.CaCarryingLine2].Cmd.bEnable:=TRUE;
							arrAxisCtrl[AxiseNo.AxisName.CaCarryingUpDown2].Cmd.bEnable:=TRUE;
							arrAxisCtrl[AxiseNo.AxisName.CaDTCarryingLine].Cmd.bEnable:=TRUE;
							arrAxisCtrl[AxiseNo.AxisName.CaDTCarryingUpDown].Cmd.bEnable:=TRUE;
							IF arrAxisCtrl[AxiseNo.AxisName.CaCarryingLine2].Status.Enabled AND arrAxisCtrl[AxiseNo.AxisName.CaCarryingUpDown2].Status.Enabled AND
								arrAxisCtrl[AxiseNo.AxisName.CaDTCarryingLine].Status.Enabled AND arrAxisCtrl[AxiseNo.AxisName.CaDTCarryingUpDown].Status.Enabled THEN
								 CaCrectCamStep0:=20;
							END_IF
								
								
						20://凸轮创建
									//fbCaCrectCamCarryingLine1.bCreatTable :=TRUE;//负极取流水线平移凸轮创建
									//fbCaCrectCamCarryingUpDown1.bCreatTable:=TRUE;//负极取流水线放片升降凸轮创建
									//fbCaCrectCamCarryingUpDown1_1.bCreatTable:=TRUE;//负极取流水线取片升降凸轮创建
									//fbCaCrectCamCarryingWhirling.bCreatTable:=TRUE;//负极取流水线旋转凸轮创建
									 fbCaCrectCamCarryingLine2.bCreatTable :=TRUE;//负极送片搬运平移凸轮创建
									 fbCaCrectCamCarryingUpDown2.bCreatTable:=TRUE;//负极送片搬运升降取片凸轮创建
									 fbCaCrectCamCarryingUpDown2_1.bCreatTable:=TRUE;//负极送片搬运升降放片凸轮创建
									 fbCaCrectCamCarryingUpDown2_3.bCreatTable:=TRUE;//负极送片搬运升降放片凸轮创建
									 fbCaCrectCamDTCarryingLine.bCreatTable :=TRUE;//负极叠片搬运平移凸轮创建
									 fbCaCrectCamDTCarryingUpDown.bCreatTable:=TRUE;//负极叠片搬运升降取片凸轮创建
									 fbCaCrectCamDTCarryingUpDown1.bCreatTable:=TRUE;//负极叠片搬运升降放片凸轮创建
									  fbCaCrectCamDTCarryingUpDown3.bCreatTable:=TRUE;//负极叠片搬运升降放片凸轮创建
									 Mach_Control.Ca_b.CreateCamDone:=FALSE;
									 CaCrectCamStep0:=30;
						30://判断凸轮是否创建完成
									IF fbCaCrectCamCarryingLine2.bCreatTableDone AND  fbCaCrectCamCarryingUpDown2.bCreatTableDone AND  fbCaCrectCamCarryingUpDown2_1.bCreatTableDone  AND
										 fbCaCrectCamDTCarryingLine.bCreatTableDone AND fbCaCrectCamDTCarryingUpDown.bCreatTableDone AND fbCaCrectCamDTCarryingUpDown1.bCreatTableDone  AND
                                        fbCaCrectCamCarryingUpDown2_3.bCreatTableDone AND  fbCaCrectCamDTCarryingUpDown3.bCreatTableDone  THEN
											Mach_Control.Ca_b.CreateCamDone:=TRUE;
											CaCrectCamStep0:=6666;
									ELSE
											IF fbCaCrectCamCarryingLine2.bCreatTableError OR fbCaCrectCamCarryingUpDown2.bCreatTableError OR fbCaCrectCamCarryingUpDown2_1.bCreatTableError  OR 
												fbCaCrectCamDTCarryingLine.bCreatTableError OR fbCaCrectCamDTCarryingUpDown.bCreatTableError OR  fbCaCrectCamDTCarryingUpDown1.bCreatTableError OR 
                                          fbCaCrectCamCarryingUpDown2_3.bCreatTableError OR  fbCaCrectCamDTCarryingUpDown3.bCreatTableError    THEN								
												Mach_Control.Ca_b.Error[0]:=TRUE;//负极取片创建凸轮报警
												CaCrectCamStep0:=9999;
											END_IF
									END_IF
				END_CASE




(***********************************负极凸轮耦合***********************************************)
(*
      fbCaCamInCarryingLine1                      :FB_CamIn ;    
      fbCaCamInCarryingUpDown1               :FB_CamIn ;    
      fbCaCamInCarryingLine2                     :FB_CamIn ;    
      fbCaCamInCarryingUpDown2              :FB_CamIn ;    
      fbCaCamInDTCarryingLine                   :FB_CamIn ;    
      fbCaCamInDTCarryingUpDown            :FB_CamIn ;    
*)

//负极取流水线搬运平移凸轮耦合
fbCaCamInCarryingLine1.ParCamIn.SlaveScaling;
fbCaCamInCarryingLine1(
	Reset:=                      stSysState.bReset  , 
	bCamInExecute:=       fbCaCamInCarryingLine1.bCamInExecute, 
	iTable1:=                   TableNo.M_CaCarryingLine1  , 
	iTable2:=                   , 
	iTableSel:=                 , 
	ParCamIn:= , 
  	axisMaster:=            arrAxis[AxiseNo.VirAxisName.CaCarryingVirGM] ,  
	axisSlave:=               arrAxis[AxiseNo.AxisName.CaCarryingLine1] ,  
	bError=> , 
	bReady=> , 
	bInSync=> );

(*Mach_Control.Ca_b.Error[11]:=*)fbCaCamInCarryingLine1.bError;
fbCaCamInCarryingLine1.bReady;
fbCaCamInCarryingLine1.bInSync;

//负极取流水线搬运升降凸轮耦合
fbCaCamInCarryingUpDown1.iTableSel;
fbCaCamInCarryingUpDown1(
	Reset:=                      stSysState.bReset  , 
	bCamInExecute:=       fbCaCamInCarryingUpDown1.bCamInExecute, 
	iTable1:=                   TableNo.M_CaCarryingUpDown1  , 
	iTable2:=                   TableNo.M_CaCarryingUpDown1_1 , 
	iTableSel:=                  , 
	ParCamIn:=                  , 
  	axisMaster:=            arrAxis[AxiseNo.VirAxisName.CaCarryingVirGM] ,  
	axisSlave:=               arrAxis[AxiseNo.AxisName.CaCarryingUpDown1] ,  
	bError=> , 
	bReady=> , 
	bInSync=> );

(*Mach_Control.Ca_b.Error[12]:=*)fbCaCamInCarryingUpDown1.bError;
fbCaCamInCarryingUpDown1.bReady;
fbCaCamInCarryingUpDown1.bInSync;
//负极取流水线旋转
fbCaCamInCarryingWhirling.ParCamIn.SlaveScaling;
fbCaCamInCarryingWhirling(
	Reset:=                      stSysState.bReset  , 
	bCamInExecute:=       fbCaCamInCarryingWhirling.bCamInExecute, 
	iTable1:=                   TableNo.M_CaCarryingWhirling1  , 
	iTable2:=                   , 
	iTableSel:=                 , 
	ParCamIn:= , 
  	axisMaster:=            arrAxis[AxiseNo.VirAxisName.CaCarryingVirGM] ,  
	axisSlave:=               arrAxis[AxiseNo.AxisName.CaCarryingWhirling1] ,  
	bError=> , 
	bReady=> , 
	bInSync=> );

fbCaCamInCarryingWhirling.bError;
fbCaCamInCarryingWhirling.bReady;
fbCaCamInCarryingWhirling.bInSync;




//负极送片搬运平移凸轮耦合
fbCaCamInCarryingLine2.ParCamIn.SlaveScaling;
fbCaCamInCarryingLine2.ParCamIn.MasterScaling:=fCaScaling;//20240508 CF
fbCaCamInCarryingLine2(
	Reset:=                      stSysState.bReset  , 
	bCamInExecute:=       fbCaCamInCarryingLine2.bCamInExecute, 
	iTable1:=                   TableNo.M_CaCarryingLine2  , 
	iTable2:=                   , 
	iTableSel:=                 , 
	ParCamIn:= , 
  	axisMaster:=            arrAxis[AxiseNo.VirAxisName.VirMain] ,  
	axisSlave:=               arrAxis[AxiseNo.AxisName.CaCarryingLine2] ,  
	bError=> , 
	bReady=> , 
	bInSync=> );
(*Mach_Control.Ca_b.Error[13]:=*)fbCaCamInCarryingLine2.bError;
fbCaCamInCarryingLine2.bReady;
fbCaCamInCarryingLine2.bInSync;


//负极送纠偏搬动升降凸轮耦合
fbCaCamInCarryingUpDown2.ParCamIn.MasterScaling:=fCaScaling;//20240508 CF
fbCaCamInCarryingUpDown2(
	Reset:=                      stSysState.bReset  , 
	bCamInExecute:=       fbCaCamInCarryingUpDown2.bCamInExecute, 
	iTable1:=                   TableNo.M_CaCarryingUpDown2  , 
	iTable2:=                   TableNo.M_CaCarryingUpDown2_1  , 
	iTable3:=                   TableNo.M_CaCarryingUpDown2_3  , 
	iTableSel:=                  , //耦合凸轮选择
	ParCamIn:=                  , 
  	axisMaster:=            arrAxis[AxiseNo.VirAxisName.VirMain] ,  
	axisSlave:=               arrAxis[AxiseNo.AxisName.CaCarryingUpDown2] ,  
	bError=> , 
	bReady=> , 
	bInSync=> );

(*Mach_Control.Ca_b.Error[14]:=*)fbCaCamInCarryingUpDown2.bError;
fbCaCamInCarryingUpDown2.bReady;
fbCaCamInCarryingUpDown2.bInSync;


//负极叠台搬运平移凸轮耦合
fbCaCamInDTCarryingLine.ParCamIn.SlaveScaling;
fbCaCamInDTCarryingLine(
	Reset:=                      stSysState.bReset  , 
	bCamInExecute:=       fbCaCamInDTCarryingLine.bCamInExecute, 
	iTable1:=                   TableNo.M_CaDTCarryingLine  , 
	iTable2:=                   , 
	iTableSel:=                 , 
	ParCamIn:=                , 
  	axisMaster:=            arrAxis[AxiseNo.VirAxisName.VirMain] ,  
	axisSlave:=               arrAxis[AxiseNo.AxisName.CaDTCarryingLine] ,  
	bError=> , 
	bReady=> , 
	bInSync=> );
(*Mach_Control.Ca_b.Error[15]:=*)fbCaCamInDTCarryingLine.bError;
fbCaCamInDTCarryingLine.bReady;
fbCaCamInDTCarryingLine.bInSync;


//负极叠台搬运升降凸轮耦合
fbCaCamInDTCarryingUpDown(
	Reset:=                      stSysState.bReset  , 
	bCamInExecute:=       fbCaCamInDTCarryingUpDown.bCamInExecute, 
	iTable1:=                   TableNo.M_CaDTCarryingUpDown  , 
	iTable2:=                    TableNo.M_CaDTCarryingUpDown1, 
	iTable3:=                    TableNo.M_CaDTCarryingUpDown3, 
	iTableSel:=                  , 
	ParCamIn:=                  , 
  	axisMaster:=            arrAxis[AxiseNo.VirAxisName.VirMain] ,  
	axisSlave:=               arrAxis[AxiseNo.AxisName.CaDTCarryingUpDown] ,  
	bError=> , 
	bReady=> , 
	bInSync=> );

(*Mach_Control.Ca_b.Error[16]:=*)fbCaCamInDTCarryingUpDown.bError;
fbCaCamInDTCarryingUpDown.bReady;
fbCaCamInDTCarryingUpDown.bInSync;


IF fbCaCamInCarryingLine1.bError OR fbCaCamInCarryingUpDown1.bError OR fbCaCamInCarryingLine2.bError OR fbCaCamInCarryingUpDown2.bError OR fbCaCamInDTCarryingLine.bError OR fbCaCamInDTCarryingUpDown.bError THEN
		Mach_Control.Ca_b.Error[11]:=TRUE;//负极藕合凸轮报警
	ELSE	
		Mach_Control.Ca_b.Error[11]:=FALSE;
END_IF
END_ACTION

ACTION Ca_Conditions:
(********************负极放弃取片********************)
Mach_Control.Ca_b.JumpPiceReady:=Mach_Control.U.DT_iMode<>1 OR Mach_Control.Ca_b.Ca_SegbeltFalg OR Mach_Control.U.EmptyRunMode OR   (Mach_Control.DT_b.SinStepMode AND Ca_StandbyStep2<>35 AND Ca_StandbyStep2<>40);

(********************负极取片准备好********************)
Mach_Control.Ca_b.GetPiceReady:=NOT Mach_Control.Ca_b.JumpPiceReady AND
														arrAxisCtrl[AxiseNo.AxisName.CaCarryingUpDown1].Status.Homed AND arrAxisCtrl[AxiseNo.AxisName.CaCarryingUpDown1].Cmd.arrbRealPoint[1] AND
														arrAxisCtrl[AxiseNo.AxisName.CaCarryingLine1].Status.Homed AND arrAxisCtrl[AxiseNo.AxisName.CaCarryingLine1].Cmd.arrbRealPoint[1];
(*
IF Mach_Control.U.DT_iMode=1 AND NOT Mach_Control.Ca_b.Ca_SegbeltFalg AND (DP_Step0<>6030 AND DP_Step0<>6040 AND 
Mach_Control.An_b.An_Quantited <= Par.stDT_date.An_Quantity  AND  Mach_Control.Ca_b.Ca_Quantited < Par.stDT_date.Ca_Quantity) AND
   arrAxisCtrl[AxiseNo.AxisName.CaCarryingUpDown1].Status.Homed AND arrAxisCtrl[AxiseNo.AxisName.CaCarryingUpDown1].Cmd.arrbRealPoint[1] AND
   arrAxisCtrl[AxiseNo.AxisName.CaCarryingLine1].Status.Homed AND arrAxisCtrl[AxiseNo.AxisName.CaCarryingLine1].Cmd.arrbRealPoint[1] THEN
 		Mach_Control.Ca_b.GetPiceReady:=TRUE;
ELSE
 		Mach_Control.Ca_b.GetPiceReady:=FALSE;	
END_IF

IF Mach_Control.U.DT_iMode<>1 OR Mach_Control.Ca_b.Ca_SegbeltFalg OR JumpPiceReady_temp1 OR JumpPiceReady_temp2 OR JumpPiceReady_temp3 THEN
	Mach_Control.Ca_b.JumpPiceReady:=TRUE;
ELSE
	Mach_Control.Ca_b.JumpPiceReady:=FALSE;
END_IF
*)



//负极纠偏平台放极片允许
IF  NOT Mach_Control.Ca_b.Ca_deviationFalg AND arrAxisCtrl[AxiseNo.AxisName.CadeviationX1].Status.Homed AND NOT arrAxisCtrl[AxiseNo.AxisName.CadeviationX1].Status.Error AND 
	arrAxisCtrl[AxiseNo.AxisName.CadeviationX1].Status.NoMoving AND arrAxisCtrl[AxiseNo.AxisName.CadeviationX1].Cmd.arrbRealPoint[1] AND 
	arrAxisCtrl[AxiseNo.AxisName.CadeviationX2].Status.Homed AND NOT arrAxisCtrl[AxiseNo.AxisName.CadeviationX2].Status.Error AND 
	arrAxisCtrl[AxiseNo.AxisName.CadeviationX2].Status.NoMoving AND arrAxisCtrl[AxiseNo.AxisName.CadeviationX2].Cmd.arrbRealPoint[1] AND 
	arrAxisCtrl[AxiseNo.AxisName.CadeviationY].Status.Homed AND NOT arrAxisCtrl[AxiseNo.AxisName.CadeviationY].Status.Error AND 
	arrAxisCtrl[AxiseNo.AxisName.CadeviationY].Status.NoMoving AND arrAxisCtrl[AxiseNo.AxisName.CadeviationY].Cmd.arrbRealPoint[1] THEN
	Mach_Control.Ca_b.Ca_deviationFPOK:=TRUE;
ELSE
	Mach_Control.Ca_b.Ca_deviationFPOK:=FALSE;	
END_IF

//负极搬运皮带取极片允许
IF  Par.stDT_date.Ca_betlCount.5 AND arrAxisCtrl[AxiseNo.AxisName.CaBelt].Status.NoMoving AND NOT arrAxisCtrl[AxiseNo.AxisName.CaBelt].Status.Error THEN
	Mach_Control.Ca_b.Ca_CacheBeltDLOK:=TRUE;
ELSE
	Mach_Control.Ca_b.Ca_CacheBeltDLOK:=FALSE;	
END_IF



//负极搬运皮带放极片允许
IF NOT  Par.stDT_date.Ca_betlCount.0 AND arrAxisCtrl[AxiseNo.AxisName.CaCarryingUpDown1].Status.NoMoving AND NOT arrAxisCtrl[AxiseNo.AxisName.CaCarryingUpDown1].Status.Error  THEN
	Mach_Control.Ca_b.Ca_CacheBeltFLOK:=TRUE;
ELSE
	Mach_Control.Ca_b.Ca_CacheBeltFLOK:=FALSE;
END_IF
//负极搬运升降1、负极搬运升降2允许负极流水线电机转动   根据实际情况修改 20240509 CF
IF ((arrAxisCtrl[AxiseNo.AxisName.CaCarryingUpDown1].Status.fSetPos <= arrAxisPar[AxiseNo.AxisName.CaCarryingUpDown1].arrTargetPoint[3]-4
	  AND arrAxisCtrl[AxiseNo.AxisName.CaCarryingUpDown1].Status.Homed ) OR
	 (arrAxisCtrl[AxiseNo.AxisName.CaCarryingLine1].Status.fActPos < arrAxisPar[AxiseNo.AxisName.CaCarryingLine1].arrTargetPoint[2]-100  
	  AND arrAxisCtrl[AxiseNo.AxisName.CaCarryingLine1].Status.Homed ) ) AND
	 
	 ((arrAxisCtrl[AxiseNo.AxisName.CaCarryingUpDown2].Status.fSetPos <= arrAxisPar[AxiseNo.AxisName.CaCarryingUpDown2].arrTargetPoint[2]-4
	   AND arrAxisCtrl[AxiseNo.AxisName.CaCarryingUpDown2].Status.Homed ) OR 
	   (arrAxisCtrl[AxiseNo.AxisName.CaCarryingLine2].Status.fActPos > arrAxisPar[AxiseNo.AxisName.CaCarryingLine2].arrTargetPoint[1]+225  
	     AND  arrAxisCtrl[AxiseNo.AxisName.CaCarryingLine2].Status.Homed ) ) THEN
	Mach_Control.Ca_b.Ca_betlMoveOK:=TRUE;
ELSE
	Mach_Control.Ca_b.Ca_betlMoveOK:=FALSE;	
END_IF


(*  南昌备份
IF ((arrAxisCtrl[AxiseNo.AxisName.CaCarryingUpDown1].Status.fSetPos <= arrAxisPar[AxiseNo.AxisName.CaCarryingUpDown1].arrTargetPoint[1]+0.5)
	 OR arrAxisCtrl[AxiseNo.AxisName.CaCarryingLine1].Cmd.arrbRealPoint[1]) AND arrAxisCtrl[AxiseNo.AxisName.CaCarryingUpDown1].Status.Homed AND
	 
	 ((arrAxisCtrl[AxiseNo.AxisName.CaCarryingUpDown2].Status.fSetPos <= arrAxisPar[AxiseNo.AxisName.CaCarryingUpDown2].arrTargetPoint[4]+0.5) 
	OR arrAxisCtrl[AxiseNo.AxisName.CaCarryingLine2].Cmd.arrbRealPoint[2]) AND arrAxisCtrl[AxiseNo.AxisName.CaCarryingUpDown1].Status.Homed  THEN
	Mach_Control.Ca_b.Ca_betlMoveOK:=TRUE;
ELSE
	Mach_Control.Ca_b.Ca_betlMoveOK:=FALSE;	
END_IF
*)


//负极搬运平移2在安全位,、负极叠片升降在安全位、尾卷夹隔膜平移在安全位、允许负极叠片搬运平移移动纠偏平台位
//arrAxisCtrl[AxiseNo.AxisName.TailCurlSEPTALine].Status.Homed  AND arrAxisCtrl[AxiseNo.AxisName.TailCurlSEPTALine].Status.fActPos <= arrAxisPar[AxiseNo.AxisName.TailCurlSEPTALine].arrTargetPoint[1] 
IF arrAxisCtrl[AxiseNo.AxisName.CaCarryingLine2].Status.Homed AND arrAxisCtrl[AxiseNo.AxisName.CaCarryingLine2].Status.NoMoving AND arrAxisCtrl[AxiseNo.AxisName.CaCarryingLine2].Cmd.arrbRealPoint[1] AND
    arrAxisCtrl[AxiseNo.AxisName.CaDTCarryingUpDown].Status.Homed AND arrAxisCtrl[AxiseNo.AxisName.CaDTCarryingUpDown].Status.NoMoving AND  TailCurlSEPTA_SafePos AND
 	 arrAxisCtrl[AxiseNo.AxisName.CaDTCarryingUpDown].Status.fSetPos   <=arrAxisPar[AxiseNo.AxisName.CaDTCarryingUpDown].arrTargetPoint[4]+0.1 THEN
	Mach_Control.Ca_b.CarryingSafepos[0]:=TRUE;
ELSE
	Mach_Control.Ca_b.CarryingSafepos[0]:=FALSE;	
END_IF
//隔膜平移在正极片位、负极叠片搬运升降在安全位，允许负极叠片搬运平移至叠片位
IF arrAxisCtrl[AxiseNo.AxisName.SEPTATLine].Status.Homed  AND arrAxisCtrl[AxiseNo.AxisName.SEPTATLine].Status.NoMoving AND arrAxisCtrl[AxiseNo.AxisName.SEPTATLine].Cmd.arrbRealPoint[1] AND 
    arrAxisCtrl[AxiseNo.AxisName.CaDTCarryingUpDown].Status.Homed AND  arrAxisCtrl[AxiseNo.AxisName.CaDTCarryingUpDown].Status.NoMoving AND arrAxisCtrl[AxiseNo.AxisName.CaDTCarryingUpDown].Cmd.arrbRealPoint[1] AND
	arrAxis[AxiseNo.AxisName.TailCurlSEPTALine].Status.Homed  AND arrAxisCtrl[AxiseNo.AxisName.TailCurlSEPTALine].Status.fSetPos <= arrAxisPar[AxiseNo.AxisName.TailCurlSEPTALine].arrTargetPoint[1]   THEN
	Mach_Control.Ca_b.CarryingSafepos[1]:=TRUE;
ELSE
	Mach_Control.Ca_b.CarryingSafepos[1]:=FALSE;
END_IF
//负极送片搬运升降2在安全位，允许负极送片搬运2平移至取流水线极片位
IF arrAxisCtrl[AxiseNo.AxisName.CaCarryingUpDown2].Cmd.arrbRealPoint[1] AND arrAxisCtrl[AxiseNo.AxisName.CaCarryingLine2].Status.Homed AND
	arrAxisCtrl[AxiseNo.AxisName.CaCarryingLine2].Status.NoMoving THEN
	Mach_Control.Ca_b.CarryingSafepos[2]:=TRUE;
ELSE
	Mach_Control.Ca_b.CarryingSafepos[2]:=FALSE;
END_IF
//负极送片搬运升降2在安全位、负极叠片搬运在安全位，允许负极送片搬运2平移至纠偏位
IF arrAxisCtrl[AxiseNo.AxisName.CaCarryingUpDown2].Cmd.arrbRealPoint[1] AND arrAxisCtrl[AxiseNo.AxisName.CaCarryingUpDown2].Status.Homed AND
	arrAxisCtrl[AxiseNo.AxisName.CaCarryingUpDown2].Status.NoMoving AND arrAxisCtrl[AxiseNo.AxisName.CaDTCarryingLine].Status.Homed  AND 
	arrAxisCtrl[AxiseNo.AxisName.CaDTCarryingLine].Status.NoMoving AND arrAxisCtrl[AxiseNo.AxisName.CaDTCarryingLine].Cmd.arrbRealPoint[2]  THEN
	Mach_Control.Ca_b.CarryingSafepos[3]:=TRUE;
ELSE
	Mach_Control.Ca_b.CarryingSafepos[3]:=FALSE;
END_IF	
//负极送片搬运升降1在安全位，允许负极搬运平移1移动
IF  arrAxisCtrl[AxiseNo.AxisName.CaCarryingUpDown1].Cmd.arrbRealPoint[1] AND arrAxisCtrl[AxiseNo.AxisName.CaCarryingUpDown1].Status.Homed AND
	arrAxisCtrl[AxiseNo.AxisName.CaCarryingUpDown1].Status.NoMoving THEN
	Mach_Control.Ca_b.CarryingSafepos[4]:=TRUE;
ELSE
	Mach_Control.Ca_b.CarryingSafepos[4]:=FALSE;
END_IF		 
//负极送片搬运安全位，负极叠片搬运安全位，尾卷夹隔膜平移，允许纠偏平台移动
IF arrAxisCtrl[AxiseNo.AxisName.CaCarryingUpDown2].Status.Homed AND arrAxisCtrl[AxiseNo.AxisName.CaCarryingLine2].Status.Homed  AND 
	(arrAxisCtrl[AxiseNo.AxisName.CaCarryingUpDown2].Status.fSetPos<=(arrAxisPar[AxiseNo.AxisName.CaCarryingUpDown2].arrTargetPoint[4]+2) OR arrAxisCtrl[AxiseNo.AxisName.CaCarryingLine2].Cmd.arrbRealPoint[1]) AND 
    arrAxisCtrl[AxiseNo.AxisName.CaDTCarryingUpDown].Status.Homed AND arrAxisCtrl[AxiseNo.AxisName.CaDTCarryingLine].Status.Homed  AND 
	(arrAxisCtrl[AxiseNo.AxisName.CaDTCarryingUpDown].Status.fSetPos<=(arrAxisPar[AxiseNo.AxisName.CaDTCarryingUpDown].arrTargetPoint[4]+2) OR arrAxisCtrl[AxiseNo.AxisName.CaDTCarryingLine].Cmd.arrbRealPoint[2]) (*AND 
	arrAxisCtrl[AxiseNo.AxisName.TailCurlSEPTALine].Status.Homed AND arrAxisCtrl[AxiseNo.AxisName.TailCurlSEPTALine].Status.fActPos<=arrAxisPar[AxiseNo.AxisName.TailCurlSEPTALine].arrTargetPoint[1]  *) THEN
	Mach_Control.Ca_b.CarryingSafepos[5]:=TRUE;
ELSE
	Mach_Control.Ca_b.CarryingSafepos[5]:=FALSE;
END_IF		
//负极取流水线机械手在安全位，允许模切流水线移动
(*
IF arrAxisCtrl[AxiseNo.AxisName.CaCarryingUpDown1].Status.Homed AND NOT Mach_Control.Ca_b.Ca_MainBelting AND 
 	(arrAxisCtrl[AxiseNo.AxisName.CaCarryingUpDown1].Status.fSetPos<=arrAxisPar[AxiseNo.AxisName.CaCarryingUpDown1].arrTargetPoint[1]+0.2 OR 
	  arrAxisCtrl[AxiseNo.AxisName.CaCarryingLine1].Cmd.arrbRealPoint[1]	) THEN
	Mach_Control.Ca_b.Ca_BeltSafe:=TRUE;
ELSE
	Mach_Control.Ca_b.Ca_BeltSafe:=FALSE;
END_IF
*)
(*
IF  Mach_Control.Ca_b.Ca_MainBelting THEN
	Mach_Control.Ca_b.Ca_BeltSafe:=TRUE;
ELSIF NOT Mach_Control.Ca_b.Ca_MainBelting AND  arrAxisCtrl[AxiseNo.AxisName.CaCarryingUpDown1].Cmd.arrbRealPoint[4] THEN
	Mach_Control.Ca_b.Ca_BeltSafe:=FALSE;
END_IF
*)
IF  Mach_Control.Ca_b.Ca_MainBelting THEN
	Mach_Control.Ca_b.Ca_BeltSafe:=TRUE;
ELSE
	Mach_Control.Ca_b.Ca_BeltSafe:=FALSE;
END_IF
//负极主流水线取片完成延时复位
Ca_BeltTon(IN:=Mach_Control.Ca_b.Ca_BeltDone , PT:=T#20MS , Q=> , ET=> );
IF Ca_BeltTon.Q THEN
	Mach_Control.Ca_b.Ca_BeltDone:=FALSE;//复位主流水线取片完成
END_IF




/////////////////////////////////////////////////////////////
/////////////////////////////////////////////////////////
////////////////////////////////////////////电机条件

//负极送片皮带
IF Mach_Control.U.DT_iMode=3  AND arrAxisCtrl[AxiseNo.AxisName.CaCarryingUpDown1].Status.fActPos<= arrAxisPar[AxiseNo.AxisName.CaCarryingUpDown1].arrTargetPoint[1] +0.5
AND  arrAxisCtrl[AxiseNo.AxisName.CaCarryingUpDown2].Status.fActPos<=arrAxisPar[AxiseNo.AxisName.CaCarryingUpDown2].arrTargetPoint[4]+0.5  THEN
	arrAxisCtrl[AxiseNo.AxisName.CaBelt].Cmd.Home_Condition:=TRUE;
	arrAxisCtrl[AxiseNo.AxisName.CaBelt].Cmd.JogN_Condition:=TRUE;
	arrAxisCtrl[AxiseNo.AxisName.CaBelt].Cmd.JogP_Condition:=TRUE;
ELSE
	arrAxisCtrl[AxiseNo.AxisName.CaBelt].Cmd.Home_Condition:=FALSE;	
	arrAxisCtrl[AxiseNo.AxisName.CaBelt].Cmd.JogN_Condition:=FALSE;
	arrAxisCtrl[AxiseNo.AxisName.CaBelt].Cmd.JogP_Condition:=FALSE;
END_IF



//负极送片搬运1平移
IF Mach_Control.U.DT_iMode=3 AND arrAxisCtrl[AxiseNo.AxisName.CaCarryingUpDown1].Status.Homed AND
 	arrAxisCtrl[AxiseNo.AxisName.CaCarryingUpDown1].Status.fSetPos<= arrAxisPar[AxiseNo.AxisName.CaCarryingUpDown1].arrTargetPoint[1]+1 THEN
	arrAxisCtrl[AxiseNo.AxisName.CaCarryingLine1].Cmd.Home_Condition:=TRUE;
ELSE
arrAxisCtrl[AxiseNo.AxisName.CaCarryingLine1].Cmd.Home_Condition:=FALSE;	
END_IF

IF Mach_Control.U.DT_iMode=3 AND arrAxisCtrl[AxiseNo.AxisName.CaCarryingLine1].Status.Homed AND 
	arrAxisCtrl[AxiseNo.AxisName.CaCarryingUpDown1].Status.Homed AND
 	arrAxisCtrl[AxiseNo.AxisName.CaCarryingUpDown1].Status.fSetPos<= arrAxisPar[AxiseNo.AxisName.CaCarryingUpDown1].arrTargetPoint[1]+1 THEN
	arrAxisCtrl[AxiseNo.AxisName.CaCarryingLine1].Cmd.GoPoint_Condition[1]:=TRUE;
ELSE
	arrAxisCtrl[AxiseNo.AxisName.CaCarryingLine1].Cmd.GoPoint_Condition[1]:=FALSE;	
END_IF

IF Mach_Control.U.DT_iMode=3 AND arrAxisCtrl[AxiseNo.AxisName.CaCarryingLine1].Status.Homed AND
	arrAxisCtrl[AxiseNo.AxisName.CaCarryingUpDown1].Status.Homed AND
 	arrAxisCtrl[AxiseNo.AxisName.CaCarryingUpDown1].Status.fSetPos<= arrAxisPar[AxiseNo.AxisName.CaCarryingUpDown1].arrTargetPoint[1]+1 THEN
		arrAxisCtrl[AxiseNo.AxisName.CaCarryingLine1].Cmd.GoPoint_Condition[2]:=TRUE;
ELSE
		arrAxisCtrl[AxiseNo.AxisName.CaCarryingLine1].Cmd.GoPoint_Condition[2]:=FALSE;	
END_IF

//负极送片搬运1升降
IF Mach_Control.U.DT_iMode=3  THEN
	arrAxisCtrl[AxiseNo.AxisName.CaCarryingUpDown1].Cmd.Home_Condition:=TRUE;
ELSE
	arrAxisCtrl[AxiseNo.AxisName.CaCarryingUpDown1].Cmd.Home_Condition:=FALSE;	
END_IF

IF Mach_Control.U.DT_iMode=3 AND arrAxisCtrl[AxiseNo.AxisName.CaCarryingUpDown1].Status.Homed THEN
	arrAxisCtrl[AxiseNo.AxisName.CaCarryingUpDown1].Cmd.GoPoint_Condition[1]:=TRUE;
ELSE
	arrAxisCtrl[AxiseNo.AxisName.CaCarryingUpDown1].Cmd.GoPoint_Condition[1]:=FALSE;	
END_IF

IF arrAxisCtrl[AxiseNo.AxisName.CaCarryingLine1].Cmd.arrbRealPoint[1] AND  Mach_Control.U.DT_iMode=3 AND arrAxisCtrl[AxiseNo.AxisName.CaCarryingUpDown1].Status.Homed THEN
	arrAxisCtrl[AxiseNo.AxisName.CaCarryingUpDown1].Cmd.GoPoint_Condition[2]:=TRUE;
ELSE
	arrAxisCtrl[AxiseNo.AxisName.CaCarryingUpDown1].Cmd.GoPoint_Condition[2]:=FALSE;	
END_IF

IF arrAxisCtrl[AxiseNo.AxisName.CaCarryingLine1].Cmd.arrbRealPoint[2] AND  Mach_Control.U.DT_iMode=3 AND arrAxisCtrl[AxiseNo.AxisName.CaCarryingUpDown1].Status.Homed THEN
	arrAxisCtrl[AxiseNo.AxisName.CaCarryingUpDown1].Cmd.GoPoint_Condition[3]:=TRUE;
ELSE
	arrAxisCtrl[AxiseNo.AxisName.CaCarryingUpDown1].Cmd.GoPoint_Condition[3]:=FALSE;	
END_IF

//负极送片搬运2平移
IF Mach_Control.U.DT_iMode=3 AND arrAxisCtrl[AxiseNo.AxisName.CaCarryingUpDown2].Status.Homed AND
 arrAxisCtrl[AxiseNo.AxisName.CaCarryingUpDown2].Status.fSetPos<=arrAxisPar[AxiseNo.AxisName.CaCarryingUpDown2].arrTargetPoint[1]+1    AND
 arrCyCtrl[arrCyNo.CylinderName.CaScrapbinUDCy].Io.DIOFFSwitch  AND	 arrCyCtrl[arrCyNo.CylinderName.CaScrapbinCy].Io.DIOnSwitch  THEN
		arrAxisCtrl[AxiseNo.AxisName.CaCarryingLine2].Cmd.Home_Condition:=TRUE;
ELSE
		arrAxisCtrl[AxiseNo.AxisName.CaCarryingLine2].Cmd.Home_Condition:=FALSE;	
END_IF

IF Mach_Control.U.DT_iMode=3 AND arrAxisCtrl[AxiseNo.AxisName.CaCarryingUpDown2].Status.Homed AND
arrAxisCtrl[AxiseNo.AxisName.CaCarryingUpDown2].Status.fSetPos<=arrAxisPar[AxiseNo.AxisName.CaCarryingUpDown2].arrTargetPoint[1]+1 AND
 arrAxisCtrl[AxiseNo.AxisName.CaCarryingLine2].Status.Homed AND
  arrCyCtrl[arrCyNo.CylinderName.CaScrapbinUDCy].Io.DIOFFSwitch AND	 arrCyCtrl[arrCyNo.CylinderName.CaScrapbinCy].Io.DIOnSwitch   THEN
arrAxisCtrl[AxiseNo.AxisName.CaCarryingLine2].Cmd.GoPoint_Condition[1]:=TRUE;
ELSE
arrAxisCtrl[AxiseNo.AxisName.CaCarryingLine2].Cmd.GoPoint_Condition[1]:=FALSE;	
END_IF

IF  Mach_Control.U.DT_iMode=3 AND arrAxisCtrl[AxiseNo.AxisName.CaCarryingUpDown2].Status.Homed AND
	 arrAxisCtrl[AxiseNo.AxisName.CaCarryingUpDown2].Status.fSetPos<=arrAxisPar[AxiseNo.AxisName.CaCarryingUpDown2].arrTargetPoint[1]+1 AND
 	arrAxisCtrl[AxiseNo.AxisName.CaCarryingLine2].Status.Homed AND  arrAxisCtrl[AxiseNo.AxisName.CaDTCarryingLine].Cmd.arrbRealPoint[2] AND
    arrCyCtrl[arrCyNo.CylinderName.CaScrapbinUDCy].Io.DIOFFSwitch AND	 arrCyCtrl[arrCyNo.CylinderName.CaScrapbinCy].Io.DIOnSwitch   THEN

	arrAxisCtrl[AxiseNo.AxisName.CaCarryingLine2].Cmd.GoPoint_Condition[2]:=TRUE;
ELSE
	arrAxisCtrl[AxiseNo.AxisName.CaCarryingLine2].Cmd.GoPoint_Condition[2]:=FALSE;	
END_IF

//负极送片搬运2升降
IF Mach_Control.U.DT_iMode=3  THEN
	arrAxisCtrl[AxiseNo.AxisName.CaCarryingUpDown2].Cmd.Home_Condition:=TRUE;
ELSE
	arrAxisCtrl[AxiseNo.AxisName.CaCarryingUpDown2].Cmd.Home_Condition:=FALSE;	
END_IF

IF Mach_Control.U.DT_iMode=3 AND arrAxisCtrl[AxiseNo.AxisName.CaCarryingUpDown2].Status.Homed THEN
	arrAxisCtrl[AxiseNo.AxisName.CaCarryingUpDown2].Cmd.GoPoint_Condition[1]:=TRUE;
ELSE
	arrAxisCtrl[AxiseNo.AxisName.CaCarryingUpDown2].Cmd.GoPoint_Condition[1]:=FALSE;	
END_IF

IF (*arrAxisCtrl[AxiseNo.AxisName.CaCarryingLine2].Cmd.arrbRealPoint[1] AND*)  Mach_Control.U.DT_iMode=3 AND arrAxisCtrl[AxiseNo.AxisName.CaCarryingUpDown2].Status.Homed THEN
	arrAxisCtrl[AxiseNo.AxisName.CaCarryingUpDown2].Cmd.GoPoint_Condition[2]:=TRUE;
ELSE
	arrAxisCtrl[AxiseNo.AxisName.CaCarryingUpDown2].Cmd.GoPoint_Condition[2]:=FALSE;	
END_IF

IF (*arrAxisCtrl[AxiseNo.AxisName.CaCarryingLine2].Cmd.arrbRealPoint[2] AND*)  Mach_Control.U.DT_iMode=3 AND arrAxisCtrl[AxiseNo.AxisName.CaCarryingUpDown1].Status.Homed THEN
	arrAxisCtrl[AxiseNo.AxisName.CaCarryingUpDown2].Cmd.GoPoint_Condition[3]:=TRUE;
ELSE
	arrAxisCtrl[AxiseNo.AxisName.CaCarryingUpDown2].Cmd.GoPoint_Condition[3]:=FALSE;	
END_IF

IF (*arrAxisCtrl[AxiseNo.AxisName.CaCarryingLine2].Cmd.arrbRealPoint[1] AND*)  Mach_Control.U.DT_iMode=3 AND arrAxisCtrl[AxiseNo.AxisName.CaCarryingUpDown2].Status.Homed THEN
	arrAxisCtrl[AxiseNo.AxisName.CaCarryingUpDown2].Cmd.GoPoint_Condition[4]:=TRUE;
ELSE
	arrAxisCtrl[AxiseNo.AxisName.CaCarryingUpDown2].Cmd.GoPoint_Condition[4]:=FALSE;	
END_IF

IF (*arrAxisCtrl[AxiseNo.AxisName.CaCarryingLine2].Cmd.arrbRealPoint[1] AND*)  Mach_Control.U.DT_iMode=3 AND arrAxisCtrl[AxiseNo.AxisName.CaCarryingUpDown2].Status.Homed THEN
	arrAxisCtrl[AxiseNo.AxisName.CaCarryingUpDown2].Cmd.GoPoint_Condition[5]:=TRUE;
ELSE
	arrAxisCtrl[AxiseNo.AxisName.CaCarryingUpDown2].Cmd.GoPoint_Condition[5]:=FALSE;	
END_IF


//负极送片搬运1旋转
IF Mach_Control.U.DT_iMode=3  AND
	arrAxisCtrl[AxiseNo.AxisName.CaCarryingUpDown1].Status.fSetPos<=arrAxisPar[AxiseNo.AxisName.CaCarryingUpDown1].arrTargetPoint[1]  THEN
	arrAxisCtrl[AxiseNo.AxisName.CaCarryingWhirling1].Cmd.Home_Condition:=TRUE;
ELSE
	arrAxisCtrl[AxiseNo.AxisName.CaCarryingWhirling1].Cmd.Home_Condition:=FALSE;	
END_IF

IF Mach_Control.U.DT_iMode=3  AND arrAxisCtrl[AxiseNo.AxisName.CaCarryingUpDown1].Cmd.arrbRealPoint[1] AND arrAxisCtrl[AxiseNo.AxisName.CaCarryingWhirling1].Status.Homed THEN
	arrAxisCtrl[AxiseNo.AxisName.CaCarryingWhirling1].Cmd.GoPoint_Condition[1]:=TRUE;
ELSE
	arrAxisCtrl[AxiseNo.AxisName.CaCarryingWhirling1].Cmd.GoPoint_Condition[1]:=FALSE;	
END_IF

IF Mach_Control.U.DT_iMode=3  AND arrAxisCtrl[AxiseNo.AxisName.CaCarryingUpDown1].Cmd.arrbRealPoint[1] AND arrAxisCtrl[AxiseNo.AxisName.CaCarryingWhirling1].Status.Homed THEN
	arrAxisCtrl[AxiseNo.AxisName.CaCarryingWhirling1].Cmd.GoPoint_Condition[2]:=TRUE;
ELSE
	arrAxisCtrl[AxiseNo.AxisName.CaCarryingWhirling1].Cmd.GoPoint_Condition[2]:=FALSE;	
END_IF


//负极纠偏平台X1
IF Mach_Control.U.DT_iMode=3  OR  (DP_Step0>=6015 AND   DP_Step0<=6041)   THEN
	arrAxisCtrl[AxiseNo.AxisName.CadeviationX1].Cmd.Home_Condition:=TRUE;
ELSE
	arrAxisCtrl[AxiseNo.AxisName.CadeviationX1].Cmd.Home_Condition:=FALSE;	
END_IF

IF Mach_Control.U.DT_iMode=3 AND arrAxisCtrl[AxiseNo.AxisName.CadeviationX1].Status.Homed THEN
	arrAxisCtrl[AxiseNo.AxisName.CadeviationX1].Cmd.GoPoint_Condition[1]:=TRUE;
ELSE
	arrAxisCtrl[AxiseNo.AxisName.CadeviationX1].Cmd.GoPoint_Condition[1]:=FALSE;	
END_IF

IF Mach_Control.U.DT_iMode=3 AND arrAxisCtrl[AxiseNo.AxisName.CadeviationX1].Status.Homed THEN
	arrAxisCtrl[AxiseNo.AxisName.CadeviationX1].Cmd.GoPoint_Condition[2]:=TRUE;
ELSE
	arrAxisCtrl[AxiseNo.AxisName.CadeviationX1].Cmd.GoPoint_Condition[2]:=FALSE;	
END_IF

IF Mach_Control.U.DT_iMode=3 AND arrAxisCtrl[AxiseNo.AxisName.CadeviationX1].Status.Homed THEN
	arrAxisCtrl[AxiseNo.AxisName.CadeviationX1].Cmd.GoPoint_Condition[3]:=TRUE;
ELSE
	arrAxisCtrl[AxiseNo.AxisName.CadeviationX1].Cmd.GoPoint_Condition[3]:=FALSE;	
END_IF

IF Mach_Control.U.DT_iMode=3 AND arrAxisCtrl[AxiseNo.AxisName.CadeviationX1].Status.Homed THEN
	arrAxisCtrl[AxiseNo.AxisName.CadeviationX1].Cmd.GoPoint_Condition[4]:=TRUE;
ELSE
	arrAxisCtrl[AxiseNo.AxisName.CadeviationX1].Cmd.GoPoint_Condition[4]:=FALSE;	
END_IF

IF Mach_Control.U.DT_iMode=3 AND arrAxisCtrl[AxiseNo.AxisName.CadeviationX1].Status.Homed THEN
	arrAxisCtrl[AxiseNo.AxisName.CadeviationX1].Cmd.GoPoint_Condition[5]:=TRUE;
ELSE
	arrAxisCtrl[AxiseNo.AxisName.CadeviationX1].Cmd.GoPoint_Condition[5]:=FALSE;	
END_IF

//负极纠偏平台X2
IF Mach_Control.U.DT_iMode=3  OR  (DP_Step0>=6015 AND   DP_Step0<=6041)    THEN
	arrAxisCtrl[AxiseNo.AxisName.CadeviationX2].Cmd.Home_Condition:=TRUE;
ELSE
	arrAxisCtrl[AxiseNo.AxisName.CadeviationX2].Cmd.Home_Condition:=FALSE;	
END_IF

IF Mach_Control.U.DT_iMode=3 AND arrAxisCtrl[AxiseNo.AxisName.CadeviationX2].Status.Homed THEN
	arrAxisCtrl[AxiseNo.AxisName.CadeviationX2].Cmd.GoPoint_Condition[1]:=TRUE;
ELSE
	arrAxisCtrl[AxiseNo.AxisName.CadeviationX2].Cmd.GoPoint_Condition[1]:=FALSE;	
END_IF

IF Mach_Control.U.DT_iMode=3 AND arrAxisCtrl[AxiseNo.AxisName.CadeviationX2].Status.Homed THEN
	arrAxisCtrl[AxiseNo.AxisName.CadeviationX2].Cmd.GoPoint_Condition[2]:=TRUE;
ELSE
	arrAxisCtrl[AxiseNo.AxisName.CadeviationX2].Cmd.GoPoint_Condition[2]:=FALSE;	
END_IF

IF Mach_Control.U.DT_iMode=3 AND arrAxisCtrl[AxiseNo.AxisName.CadeviationX2].Status.Homed THEN
	arrAxisCtrl[AxiseNo.AxisName.CadeviationX2].Cmd.GoPoint_Condition[3]:=TRUE;
ELSE
	arrAxisCtrl[AxiseNo.AxisName.CadeviationX2].Cmd.GoPoint_Condition[3]:=FALSE;	
END_IF

IF Mach_Control.U.DT_iMode=3 AND arrAxisCtrl[AxiseNo.AxisName.CadeviationX2].Status.Homed THEN
	arrAxisCtrl[AxiseNo.AxisName.CadeviationX2].Cmd.GoPoint_Condition[4]:=TRUE;
ELSE
	arrAxisCtrl[AxiseNo.AxisName.CadeviationX2].Cmd.GoPoint_Condition[4]:=FALSE;	
END_IF

IF Mach_Control.U.DT_iMode=3 AND arrAxisCtrl[AxiseNo.AxisName.CadeviationX2].Status.Homed THEN
	arrAxisCtrl[AxiseNo.AxisName.CadeviationX2].Cmd.GoPoint_Condition[5]:=TRUE;
ELSE
	arrAxisCtrl[AxiseNo.AxisName.CadeviationX2].Cmd.GoPoint_Condition[5]:=FALSE;	
END_IF

//负极纠偏平台Y
IF Mach_Control.U.DT_iMode=3  OR  (DP_Step0>=6015 AND   DP_Step0<=6041)  THEN
	arrAxisCtrl[AxiseNo.AxisName.CadeviationY].Cmd.Home_Condition:=TRUE;
ELSE
	arrAxisCtrl[AxiseNo.AxisName.CadeviationY].Cmd.Home_Condition:=FALSE;	
END_IF

IF Mach_Control.U.DT_iMode=3 AND arrAxisCtrl[AxiseNo.AxisName.CadeviationY].Status.Homed THEN
	arrAxisCtrl[AxiseNo.AxisName.CadeviationY].Cmd.GoPoint_Condition[1]:=TRUE;
ELSE
	arrAxisCtrl[AxiseNo.AxisName.CadeviationY].Cmd.GoPoint_Condition[1]:=FALSE;	
END_IF

IF Mach_Control.U.DT_iMode=3 AND arrAxisCtrl[AxiseNo.AxisName.CadeviationY].Status.Homed THEN
	arrAxisCtrl[AxiseNo.AxisName.CadeviationY].Cmd.GoPoint_Condition[2]:=TRUE;
ELSE
	arrAxisCtrl[AxiseNo.AxisName.CadeviationY].Cmd.GoPoint_Condition[2]:=FALSE;	
END_IF

IF Mach_Control.U.DT_iMode=3 AND arrAxisCtrl[AxiseNo.AxisName.CadeviationY].Status.Homed THEN
	arrAxisCtrl[AxiseNo.AxisName.CadeviationY].Cmd.GoPoint_Condition[3]:=TRUE;
ELSE
	arrAxisCtrl[AxiseNo.AxisName.CadeviationY].Cmd.GoPoint_Condition[3]:=FALSE;	
END_IF

IF Mach_Control.U.DT_iMode=3 AND arrAxisCtrl[AxiseNo.AxisName.CadeviationY].Status.Homed THEN
	arrAxisCtrl[AxiseNo.AxisName.CadeviationY].Cmd.GoPoint_Condition[4]:=TRUE;
ELSE
	arrAxisCtrl[AxiseNo.AxisName.CadeviationY].Cmd.GoPoint_Condition[4]:=FALSE;	
END_IF

IF Mach_Control.U.DT_iMode=3 AND arrAxisCtrl[AxiseNo.AxisName.CadeviationY].Status.Homed THEN
	arrAxisCtrl[AxiseNo.AxisName.CadeviationY].Cmd.GoPoint_Condition[5]:=TRUE;
ELSE
	arrAxisCtrl[AxiseNo.AxisName.CadeviationY].Cmd.GoPoint_Condition[5]:=FALSE;	
END_IF

//负极叠台搬运平移1
IF Mach_Control.U.DT_iMode=3 AND arrAxisCtrl[AxiseNo.AxisName.CaDTCarryingUpDown].Status.Homed AND 
	(*arrAxisCtrl[AxiseNo.AxisName.CaDTCarryingUpDown].Status.fSetPos<=arrAxisPar[AxiseNo.AxisName.CaDTCarryingUpDown].arrTargetPoint[1] AND*)
	arrAxisCtrl[AxiseNo.AxisName.CaDTCarryingUpDown].Cmd.arrbRealPoint[1] AND
	 arrAxisCtrl[AxiseNo.AxisName.CaCarryingLine2].Status.fSetPos<= arrAxisPar[AxiseNo.AxisName.CaCarryingLine2].arrTargetPoint[1]+1 AND
	//  arrAxisCtrl[AxiseNo.AxisName.SEPTATLine].Cmd.arrbRealPoint[1] AND 
		arrAxisCtrl[AxiseNo.AxisName.CaCarryingLine2].Status.Homed AND arrAxisCtrl[AxiseNo.AxisName.CaCarryingLine2].Status.NoMoving  AND
         arrCyCtrl[arrCyNo.CylinderName.CaScrapbinUDCy].Io.DIOFFSwitch  AND	 arrCyCtrl[arrCyNo.CylinderName.CaScrapbinCy].Io.DIOnSwitch THEN
	arrAxisCtrl[AxiseNo.AxisName.CaDTCarryingLine].Cmd.Home_Condition:=TRUE;
ELSE
	arrAxisCtrl[AxiseNo.AxisName.CaDTCarryingLine].Cmd.Home_Condition:=FALSE;	
END_IF

IF Mach_Control.U.WJ_iMode=3 
AND arrCyCtrl[arrCyNo.CylinderName.CaScrapbinUDCy].Status.OFFState 
AND arrCyCtrl[arrCyNo.CylinderName.CaScrapbinCy].Status.ONState THEN
   arrAxisCtrl[AxiseNo.AxisName.CaDTCarryingLine].Cmd.JogP_Condition:=TRUE;
   arrAxisCtrl[AxiseNo.AxisName.CaDTCarryingLine].Cmd.JogN_Condition:=TRUE;
   ELSE 
   arrAxisCtrl[AxiseNo.AxisName.CaDTCarryingLine].Cmd.JogP_Condition:=FALSE;
   arrAxisCtrl[AxiseNo.AxisName.CaDTCarryingLine].Cmd.JogN_Condition:=FALSE;
 END_IF


IF Mach_Control.U.DT_iMode=3 AND arrAxisCtrl[AxiseNo.AxisName.CaDTCarryingUpDown].Status.Homed AND 
 	(*arrAxisCtrl[AxiseNo.AxisName.CaDTCarryingUpDown].Status.fSetPos<=arrAxisPar[AxiseNo.AxisName.CaDTCarryingUpDown].arrTargetPoint[1] AND *)
	arrAxisCtrl[AxiseNo.AxisName.CaDTCarryingUpDown].Cmd.arrbRealPoint[1] AND
	arrAxisCtrl[AxiseNo.AxisName.CaDTCarryingLine].Status.Homed AND  arrAxisCtrl[AxiseNo.AxisName.CaCarryingLine2].Cmd.arrbRealPoint[1] 
   AND arrCyCtrl[arrCyNo.CylinderName.CaScrapbinUDCy].Status.OFFState 
   AND	 arrCyCtrl[arrCyNo.CylinderName.CaScrapbinCy].Status.ONState  THEN
	arrAxisCtrl[AxiseNo.AxisName.CaDTCarryingLine].Cmd.GoPoint_Condition[1]:=TRUE;
ELSE
	arrAxisCtrl[AxiseNo.AxisName.CaDTCarryingLine].Cmd.GoPoint_Condition[1]:=FALSE;	
END_IF


IF Mach_Control.U.DT_iMode=3 AND arrAxisCtrl[AxiseNo.AxisName.CaDTCarryingUpDown].Status.Homed
 (*arrAxisCtrl[AxiseNo.AxisName.CaDTCarryingUpDown].Status.fActPos=arrAxisPar[AxiseNo.AxisName.CaDTCarryingUpDown].arrTargetPoint[1] *)
AND  arrAxisCtrl[AxiseNo.AxisName.CaDTCarryingUpDown].Cmd.arrbRealPoint[1]
AND arrAxisCtrl[AxiseNo.AxisName.CaDTCarryingLine].Status.Homed AND arrAxisCtrl[AxiseNo.AxisName.SEPTATLine].Cmd.arrbRealPoint[1]
AND NOT arrAxisCtrl[AxiseNo.AxisName.CaDTCarryingUpDown].Cmd.arrbRealPoint[5] 
AND arrCyCtrl[arrCyNo.CylinderName.CaScrapbinUDCy].Status.OFFState 
AND	 arrCyCtrl[arrCyNo.CylinderName.CaScrapbinCy].Status.ONState  THEN
	arrAxisCtrl[AxiseNo.AxisName.CaDTCarryingLine].Cmd.GoPoint_Condition[2]:=TRUE;
ELSE
	arrAxisCtrl[AxiseNo.AxisName.CaDTCarryingLine].Cmd.GoPoint_Condition[2]:=FALSE;	
END_IF


//负极叠台搬升降移1
IF Mach_Control.U.DT_iMode=3  THEN
	arrAxisCtrl[AxiseNo.AxisName.CaDTCarryingUpDown].Cmd.Home_Condition:=TRUE;
ELSE
	arrAxisCtrl[AxiseNo.AxisName.CaDTCarryingUpDown].Cmd.Home_Condition:=FALSE;	
END_IF

IF Mach_Control.U.DT_iMode=3 AND arrAxisCtrl[AxiseNo.AxisName.CaDTCarryingUpDown].Status.Homed THEN
	arrAxisCtrl[AxiseNo.AxisName.CaDTCarryingUpDown].Cmd.GoPoint_Condition[1]:=TRUE;
ELSE
	arrAxisCtrl[AxiseNo.AxisName.CaDTCarryingUpDown].Cmd.GoPoint_Condition[1]:=FALSE;	
END_IF

IF Mach_Control.U.DT_iMode=3 AND  arrAxisCtrl[AxiseNo.AxisName.CaDTCarryingUpDown].Status.Homed THEN
	arrAxisCtrl[AxiseNo.AxisName.CaDTCarryingUpDown].Cmd.GoPoint_Condition[2]:=TRUE;
ELSE
	arrAxisCtrl[AxiseNo.AxisName.CaDTCarryingUpDown].Cmd.GoPoint_Condition[2]:=FALSE;	
END_IF

IF Mach_Control.U.DT_iMode=3 AND  arrAxisCtrl[AxiseNo.AxisName.CaDTCarryingUpDown].Status.Homed THEN
	arrAxisCtrl[AxiseNo.AxisName.CaDTCarryingUpDown].Cmd.GoPoint_Condition[3]:=TRUE;
ELSE
	arrAxisCtrl[AxiseNo.AxisName.CaDTCarryingUpDown].Cmd.GoPoint_Condition[3]:=FALSE;	
END_IF

IF Mach_Control.U.DT_iMode=3  AND arrAxisCtrl[AxiseNo.AxisName.CaDTCarryingUpDown].Status.Homed THEN
	arrAxisCtrl[AxiseNo.AxisName.CaDTCarryingUpDown].Cmd.GoPoint_Condition[4]:=TRUE;
ELSE
	arrAxisCtrl[AxiseNo.AxisName.CaDTCarryingUpDown].Cmd.GoPoint_Condition[4]:=FALSE;	
END_IF

IF Mach_Control.U.DT_iMode=3 AND arrAxisCtrl[AxiseNo.AxisName.CaDTCarryingUpDown].Status.Homed THEN
	arrAxisCtrl[AxiseNo.AxisName.CaDTCarryingUpDown].Cmd.GoPoint_Condition[5]:=TRUE;
ELSE
	arrAxisCtrl[AxiseNo.AxisName.CaDTCarryingUpDown].Cmd.GoPoint_Condition[5]:=FALSE;	
END_IF

//负极NG料盒伸缩气缸条件CaCarryingUpDown1
IF arrAxisCtrl[AxiseNo.AxisName.CaDTCarryingUpDown].Cmd.arrbRealPoint[5] AND (arrAxisCtrl[AxiseNo.AxisName.CaCarryingUpDown2].Cmd.arrbRealPoint[5] OR arrAxisCtrl[AxiseNo.AxisName.CaCarryingLine2].Cmd.arrbRealPoint[1] )
   AND  arrCyCtrl[arrCyNo.CylinderName.CaScrapbinUDCy].Io.DIOnSwitch THEN
	arrCyCtrl[arrCyNo.CylinderName.	CaScrapbinCy].Cmd.OnCondition:=TRUE;
    arrCyCtrl[arrCyNo.CylinderName.	CaScrapbinCy].Cmd.OffCondition:=TRUE;
ELSE	
	arrCyCtrl[arrCyNo.CylinderName.	CaScrapbinCy].Cmd.OnCondition:=FALSE;
    arrCyCtrl[arrCyNo.CylinderName.	CaScrapbinCy].Cmd.OffCondition:=FALSE;
END_IF
END_ACTION

ACTION Ca_Gohome:
	Ca_GohomeTon(IN:= , PT:=T#1S , Q=> , ET=> );//负极回原点延时
Ca_GohomeOverTon(IN:= , PT:=T#90S , Q=> , ET=> );//负极回原点超时报警延时
Ca_BeltGohomeOverTon(IN:= , PT:=T#90S , Q=> , ET=> );//负极皮带回原点超时报警延时
rCa_Gohome_TRIG(CLK:=Mach_Control.Ca_b.Ca_GohomeHMI , Q=> );//负极回原点启动
fCa_Gohome_TRIG(CLK:=Mach_Control.Ca_b.Ca_GohomeHMI , Q=> );//负极回原点启动


Ca_BeltGohomeTon(IN:= , PT:=T#1S , Q=> , ET=> );//负极回原点延时
Ca_BeltGohomeOverTon(IN:= , PT:=T#90S , Q=> , ET=> );//负极回原点超时报警延时
rCa_BeltGohome_TRIG(CLK:=Mach_Control.Ca_b.Ca_BeltGohomeHMI , Q=> );//
fCa_BeltGohome_TRIG(CLK:=Mach_Control.Ca_b.Ca_BeltGohomeHMI , Q=> );//

//判断回原点是否完成
		IF arrAxisCtrl[AxiseNo.AxisName.CaCarryingUpDown2].Status.Homed AND arrAxisCtrl[AxiseNo.AxisName.CaDTCarryingUpDown].Status.Homed AND 
			arrAxisCtrl[AxiseNo.AxisName.CaCarryingLine2].Status.Homed AND 	arrAxisCtrl[AxiseNo.AxisName.CadeviationX1].Status.Homed AND
			arrAxisCtrl[AxiseNo.AxisName.CadeviationX2].Status.Homed AND 	arrAxisCtrl[AxiseNo.AxisName.CadeviationY].Status.Homed AND 
			arrAxisCtrl[AxiseNo.AxisName.CaDTCarryingLine].Status.Homed AND Ca_GohomeDone THEN
					Mach_Control.Ca_b.Ca_GohomeDone:=TRUE;//负极取片回原点完成
		ELSE
					Mach_Control.Ca_b.Ca_GohomeDone:=FALSE;//负极取片回原点完成
		END_IF	
//判断负极皮带初始化是否完成
IF arrAxisCtrl[AxiseNo.AxisName.CaCarryingUpDown1].Status.Homed  AND arrAxisCtrl[AxiseNo.AxisName.CaCarryingWhirling1].Status.Homed AND 
	arrAxisCtrl[AxiseNo.AxisName.CaCarryingLine1].Status.Homed AND Ca_BeltGohomeDone THEN
		Mach_Control.Ca_b.Ca_BeltGohomeDone:=TRUE;
ELSE
		Mach_Control.Ca_b.Ca_BeltGohomeDone:=FALSE;
END_IF
 
		
		
		
		
IF Mach_Control.U.DT_iMode=3 THEN//在手动状态下
//回原点超时报警	
IF  Ca_Gohoming THEN
		IF 	NOT Ca_GohomeOverTon.Q THEN
			    Ca_GohomeOverTon.IN:=TRUE;
		ELSE
			IF 	 Ca_GohomeOverTon.Q THEN
				Ca_Gohoming:=FALSE;
			     Mach_Control.Ca_b.Error[19]:=TRUE;//负极回原点超时报警
			     Ca_GohomeOverTon.IN:=FALSE;
			END_IF	 
				 
		END_IF

ELSE
		Ca_GohomeOverTon.IN:=FALSE;
END_IF

//手动触发
IF rCa_Gohome_TRIG.Q THEN
Step_InitCaDT:=0;
Ca_GohomeDone:=FALSE;//负极取片回原点完成
Ca_Gohoming:=FALSE;//负极取片回原点中
END_IF	
//负极取料机构初始化
CASE Step_InitCaDT OF
0://等待负极回原点启动信号
	IF fCa_Gohome_TRIG.Q THEN
		Ca_GohomeDone:=FALSE;//负极取片回原点完成
		Ca_Gohoming:=TRUE;//负极取片回原点中
		Mach_Control.Ca_b.Ca_GohomeHMI:=FALSE;
		Step_InitCaDT:=1;
	END_IF	
1://复位回原点完成
	Ca_GohomeTon.IN:=FALSE;
	Mach_Control.Ca_b.Ca_MainBelting:=FALSE;
	IF NOT Ca_GohomeDone THEN
		Step_InitCaDT:=10;
	END_IF 				
10://
	Mach_Control.Ca_b.Ca_CarryingFalg:=FALSE;//负极搬运升降有料标记
	Mach_Control.Ca_b.Ca_DPCarryingFalg:=FALSE;//负极叠片搬运有料标记
	Mach_Control.Ca_b.Ca_deviationFalg:=FALSE;//负极纠偏平台有料标记
	Ca_Step0:=0;//负极搬运子程序1
	Ca_Step1:=0;//负极搬运子程序2
	Ca_Step2:=0;//负极搬运子程序3
	Ca_Step3:=0;//负极搬运子程序4
	Ca_RectifydevStep :=0;//纠偏自动程序
	Ca_Demarcate_Step0:=0;//纠偏标定程序步
	Ca_RecdevPla_Step0:=0;//纠偏自动程序步
	Ca_StandbyStep0:=0;//负极自动备料自动步清零
	Ca_StandbyStep1:=0;//叠负极片，判断真空阀的开关
	Ca_StandbyStep5:=0;//叠负极片，判断主轴是否完成
	Step_InitCaDT:=20;//取负极片回原点
20:
	//fbCaCamInCarryingLine1.bCamInExecute,:=TURE;//负极取流水线平移
	//fbCaCamInCarryingUpDown1.bCamInExecute:=TRUE;//负极取流水线升降
	fbCaCamInCarryingLine2.bCamInExecute:=FALSE;//负极送片搬运平移
	fbCaCamInCarryingUpDown2.bCamInExecute:=FALSE;//负极送片搬运升降
	fbCaCamInDTCarryingLine.bCamInExecute:=FALSE;//负极叠片搬运平移
	fbCaCamInDTCarryingUpDown.bCamInExecute:=FALSE;//负极叠片搬运升降		
	
	IF NOT fbCaCamInCarryingLine2.bCamInExecute AND NOT  fbCaCamInCarryingUpDown2.bCamInExecute AND
		 NOT fbCaCamInDTCarryingLine.bCamInExecute AND NOT  fbCaCamInDTCarryingUpDown.bCamInExecute THEN
			Step_InitCaDT:=25;
	END_IF						
25:
	arrAxisCtrl[AxiseNo.AxisName.CaCarryingUpDown1].Cmd.bHalt:=TRUE;//负极送片搬运1升降解耦
	arrAxisCtrl[AxiseNo.AxisName.CaCarryingUpDown2].Cmd.bHalt:=TRUE;//负极送片搬运2升降解耦
	arrAxisCtrl[AxiseNo.AxisName.CaDTCarryingUpDown].Cmd.bHalt:=TRUE;//负极叠台搬运升降解耦
	arrAxisCtrl[AxiseNo.AxisName.CaCarryingLine1].Cmd.bHalt:=TRUE;//负极搬运平移1解耦
	arrAxisCtrl[AxiseNo.AxisName.CaCarryingLine2].Cmd.bHalt:=TRUE;//负极搬运平移2解耦
	arrAxisCtrl[AxiseNo.AxisName.CaDTCarryingLine].Cmd.bHalt:=TRUE;//负极叠片搬运平移解耦	

	IF  NOT arrAxisCtrl[AxiseNo.AxisName.CaCarryingUpDown1].Status.Coupled AND arrAxisCtrl[AxiseNo.AxisName.CaCarryingUpDown1].Status.NoMoving AND  
	NOT arrAxisCtrl[AxiseNo.AxisName.CaCarryingUpDown2].Status.Coupled AND arrAxisCtrl[AxiseNo.AxisName.CaCarryingUpDown2].Status.NoMoving AND 
	NOT arrAxisCtrl[AxiseNo.AxisName.CaDTCarryingUpDown].Status.Coupled AND arrAxisCtrl[AxiseNo.AxisName.CaDTCarryingUpDown].Status.NoMoving AND  
	NOT arrAxisCtrl[AxiseNo.AxisName.CaCarryingLine1].Status.Coupled AND arrAxisCtrl[AxiseNo.AxisName.CaCarryingLine1].Status.NoMoving AND
	NOT arrAxisCtrl[AxiseNo.AxisName.CaCarryingLine2].Status.Coupled AND arrAxisCtrl[AxiseNo.AxisName.CaCarryingLine2].Status.NoMoving AND  
	NOT arrAxisCtrl[AxiseNo.AxisName.CaDTCarryingLine].Status.Coupled AND arrAxisCtrl[AxiseNo.AxisName.CaDTCarryingLine].Status.NoMoving THEN
		arrAxisCtrl[AxiseNo.AxisName.CaCarryingUpDown1].Cmd.bHalt:=FALSE;//负极送片搬运1升降解耦
		arrAxisCtrl[AxiseNo.AxisName.CaCarryingUpDown2].Cmd.bHalt:=FALSE;//负极送片搬运2升降解耦
		arrAxisCtrl[AxiseNo.AxisName.CaDTCarryingUpDown].Cmd.bHalt:=FALSE;//负极叠台搬运升降解耦
		arrAxisCtrl[AxiseNo.AxisName.CaCarryingLine1].Cmd.bHalt:=FALSE;//负极搬运平移1解耦
		arrAxisCtrl[AxiseNo.AxisName.CaCarryingLine2].Cmd.bHalt:=FALSE;//负极搬运平移2解耦
		arrAxisCtrl[AxiseNo.AxisName.CaDTCarryingLine].Cmd.bHalt:=FALSE;//负极叠片搬运平移解耦							   
		Step_InitCaDT:=30;
	END_IF
30://
	arrAxisCtrl[AxiseNo.AxisName.CaCarryingUpDown2].Cmd.bEnable:=TRUE;//负极送片搬运2升降
	arrAxisCtrl[AxiseNo.AxisName.CaDTCarryingUpDown].Cmd.bEnable:=TRUE;//负极叠台搬运升降
	arrAxisCtrl[AxiseNo.AxisName.CaCarryingLine2].Cmd.bEnable:=TRUE;//负极搬运平移2
	arrAxisCtrl[AxiseNo.AxisName.CaDTCarryingLine].Cmd.bEnable:=TRUE;//负极叠片搬运平移
	arrAxisCtrl[AxiseNo.AxisName.CadeviationX1].Cmd.bEnable:=TRUE;//负极纠偏X1轴使能
	arrAxisCtrl[AxiseNo.AxisName.CadeviationX2].Cmd.bEnable:=TRUE;//负极纠偏X2轴使能	
	arrAxisCtrl[AxiseNo.AxisName.CadeviationY].Cmd.bEnable:=TRUE;//负极纠偏Y轴使能		
	IF    	arrAxisCtrl[AxiseNo.AxisName.CaCarryingUpDown2].Status.Enabled AND 
		arrAxisCtrl[AxiseNo.AxisName.CaDTCarryingUpDown].Status.Enabled AND 								   
		arrAxisCtrl[AxiseNo.AxisName.CaCarryingLine2].Status.Enabled AND 
		arrAxisCtrl[AxiseNo.AxisName.CaDTCarryingLine].Status.Enabled AND 
		arrAxisCtrl[AxiseNo.AxisName.CadeviationX1].Status.Enabled AND 
		arrAxisCtrl[AxiseNo.AxisName.CadeviationX2].Status.Enabled  AND 
		arrAxisCtrl[AxiseNo.AxisName.CadeviationY].Status.Enabled  THEN
				Step_InitCaDT:=35;
	ELSIF  arrAxisCtrl[AxiseNo.AxisName.CaCarryingUpDown2].Status.Error OR 
		arrAxisCtrl[AxiseNo.AxisName.CaDTCarryingUpDown].Status.Error OR 								   
		arrAxisCtrl[AxiseNo.AxisName.CaCarryingLine2].Status.Error OR 
		arrAxisCtrl[AxiseNo.AxisName.CaDTCarryingLine].Status.Error OR 
		arrAxisCtrl[AxiseNo.AxisName.CadeviationX1].Status.Error OR 
		arrAxisCtrl[AxiseNo.AxisName.CadeviationX2].Status.Error  OR 
		arrAxisCtrl[AxiseNo.AxisName.CadeviationY].Status.Error  THEN
		Step_InitCaDT:=9999;								
	END_IF		

35://负极取片1升降，负极送片1升降、负极叠片升降回原点
	arrAxisCtrl[AxiseNo.AxisName.CaCarryingUpDown2].Cmd.bHome:=TRUE;//负极送片搬运2升降回原点	
	arrAxisCtrl[AxiseNo.AxisName.CaDTCarryingUpDown].Cmd.bHome:=TRUE;//负极叠台搬运升降回原点				
	Step_InitCaDT:=40;

40://判断回原点是否完成 arrAxisCtrl[AxiseNo.AxisName.CaCarryingUpDown1].Status.Homed AND
	IF NOT Ca_GohomeTon.Q THEN	
		Ca_GohomeTon.IN:=TRUE;
	ELSE		
		IF  arrAxisCtrl[AxiseNo.AxisName.CaCarryingUpDown2].Status.Homed AND arrAxisCtrl[AxiseNo.AxisName.CaCarryingUpDown2].Status.NoMoving AND 
			arrAxisCtrl[AxiseNo.AxisName.CaDTCarryingUpDown].Status.Homed AND arrAxisCtrl[AxiseNo.AxisName.CaDTCarryingUpDown].Status.NoMoving THEN
			arrAxisCtrl[AxiseNo.AxisName.CaCarryingUpDown2].Cmd.bHome:=FALSE;//负极送片搬运2升降回原点	
			arrAxisCtrl[AxiseNo.AxisName.CaDTCarryingUpDown].Cmd.bHome:=FALSE;//负极叠台搬运升降回原点		
			Ca_GohomeTon.IN:=FALSE;					   
			Step_InitCaDT:=45;
		ELSIF arrAxisCtrl[AxiseNo.AxisName.CaCarryingUpDown2].Status.Error OR arrAxisCtrl[AxiseNo.AxisName.CaDTCarryingUpDown].Status.Error THEN
			arrAxisCtrl[AxiseNo.AxisName.CaCarryingUpDown2].Cmd.bHome:=FALSE;//负极送片搬运2升降回原点	
			arrAxisCtrl[AxiseNo.AxisName.CaDTCarryingUpDown].Cmd.bHome:=FALSE;//负极叠台搬运升降回原点	
			Ca_GohomeTon.IN:=FALSE;	
			Ca_Gohoming:=FALSE;//负极取片回原点中	
			Step_InitCaDT:=9999;
		END_IF
	END_IF

45:
	IF arrAxisCtrl[AxiseNo.AxisName.CaCarryingUpDown2].Status.Homed AND arrAxisCtrl[AxiseNo.AxisName.CaCarryingUpDown2].Status.NoMoving THEN
		IF arrAxisCtrl[AxiseNo.AxisName.CaCarryingUpDown2].Cmd.arrbRealPoint[5] THEN
			arrAxisCtrl[AxiseNo.AxisName.CaCarryingUpDown2].Cmd.iGoSetPos:=0;
		ELSE
			arrAxisCtrl[AxiseNo.AxisName.CaCarryingUpDown2].Cmd.iGoSetPos:=5;
		END_IF	
	END_IF

	IF arrAxisCtrl[AxiseNo.AxisName.CaDTCarryingUpDown].Status.Homed AND arrAxisCtrl[AxiseNo.AxisName.CaDTCarryingUpDown].Status.NoMoving THEN
		IF arrAxisCtrl[AxiseNo.AxisName.CaDTCarryingUpDown].Cmd.arrbRealPoint[5]  THEN
			arrAxisCtrl[AxiseNo.AxisName.CaDTCarryingUpDown].Cmd.iGoSetPos:=0;
		ELSE
		   arrAxisCtrl[AxiseNo.AxisName.CaDTCarryingUpDown].Cmd.iGoSetPos:=5;
		END_IF	
	END_IF		
	
  IF arrAxisCtrl[AxiseNo.AxisName.CaCarryingUpDown2].Cmd.arrbRealPoint[5] AND arrAxisCtrl[AxiseNo.AxisName.CaDTCarryingUpDown].Cmd.arrbRealPoint[5]  THEN
	Step_InitCaDT:=50;
  END_IF	
  
	IF  arrAxisCtrl[AxiseNo.AxisName.CaDTCarryingUpDown].Status.Error OR arrAxisCtrl[AxiseNo.AxisName.CaCarryingUpDown2].Status.Error THEN
		Ca_Gohoming:=FALSE;//负极取片回原点中	
		Step_InitCaDT:=9999;
	END_IF	

	
50:
IF arrAxisCtrl[AxiseNo.AxisName.CaDTCarryingUpDown].Cmd.arrbRealPoint[5] OR arrCyCtrl[arrCyNo.CylinderName.CaScrapbinCy].Io.DIOnSwitch THEN
	arrCyCtrl[arrCyNo.CylinderName.CaScrapbinCy].Cmd.bON:=TRUE;//负极纠偏NG料盒气缸伸出
	IF arrCyCtrl[arrCyNo.CylinderName.CaScrapbinCy].Status.ONState THEN
		arrCyCtrl[arrCyNo.CylinderName.CaScrapbinUDCy].Cmd.bOFF:=TRUE;//负极纠偏NG料盒气缸升降气缸下降
		IF  arrCyCtrl[arrCyNo.CylinderName.CaScrapbinUDCy].Status.OFFState THEN								
			Step_InitCaDT:=60;
		END_IF
	ELSIF  arrCyCtrl[arrCyNo.CylinderName.CaScrapbinCy].Status.Error1 OR arrCyCtrl[arrCyNo.CylinderName.CaScrapbinCy].Status.Error2 OR
		arrCyCtrl[arrCyNo.CylinderName.CaScrapbinUDCy].Status.Error1 OR arrCyCtrl[arrCyNo.CylinderName.CaScrapbinUDCy].Status.Error2 THEN
		Ca_Gohoming:=FALSE;//负极取片回原点中	
		Step_InitCaDT:=9999;
	END_IF
ELSE
	Mach_Control.Ca_b.Error[42] :=TRUE;//负极机械手初始化时，叠台搬运升降不在避让位
	Ca_Gohoming:=FALSE;//负极取片回原点中	
	Step_InitAnDT:=9999;
END_IF
	
60:
	IF arrAxisCtrl[AxiseNo.AxisName.CaDTCarryingUpDown].Status.Homed AND arrAxisCtrl[AxiseNo.AxisName.CaDTCarryingUpDown].Status.NoMoving THEN
		IF arrAxisCtrl[AxiseNo.AxisName.CaDTCarryingUpDown].Cmd.arrbRealPoint[1]  THEN
			arrAxisCtrl[AxiseNo.AxisName.CaDTCarryingUpDown].Cmd.iGoSetPos:=0;
			Step_InitCaDT:=65;
		ELSE
		   arrAxisCtrl[AxiseNo.AxisName.CaDTCarryingUpDown].Cmd.iGoSetPos:=1;
		END_IF	
	END_IF		
	IF  arrAxisCtrl[AxiseNo.AxisName.CaDTCarryingUpDown].Status.Error THEN
		Ca_Gohoming:=FALSE;//负极取片回原点中	
		Step_InitCaDT:=9999;
	END_IF	


65://负极搬运平移1、负极搬运平移2、负极叠片平移回原点、纠偏X1轴回原点、纠偏X2轴回原点、纠偏Y轴回原点
	arrAxisCtrl[AxiseNo.AxisName.CaCarryingLine2].Cmd.bHome:=TRUE;//负极搬运平移2							
	arrAxisCtrl[AxiseNo.AxisName.CadeviationX1].Cmd.bHome:=TRUE;//负极纠偏X1
	arrAxisCtrl[AxiseNo.AxisName.CadeviationX2].Cmd.bHome:=TRUE;//负极纠偏X2
	arrAxisCtrl[AxiseNo.AxisName.CadeviationY].Cmd.bHome:=TRUE;//负极纠偏Y
	Ca_Carrying2TorMark:=TRUE;//负极搬运2平移力矩判断标志位
	Step_InitCaDT:=70;
70://判断回原点是否完成  arrAxisCtrl[AxiseNo.AxisName.CaCarryingLine1].Status.Homed AND 
	IF NOT Ca_GohomeTon.Q THEN				 
		Ca_GohomeTon.IN:=TRUE;
	ELSE			
		IF arrAxisCtrl[AxiseNo.AxisName.CaCarryingLine2].Status.Homed AND arrAxisCtrl[AxiseNo.AxisName.CaCarryingLine2].Status.NoMoving AND
			arrAxisCtrl[AxiseNo.AxisName.CadeviationX1].Status.Homed  AND arrAxisCtrl[AxiseNo.AxisName.CadeviationX1].Status.NoMoving AND
			arrAxisCtrl[AxiseNo.AxisName.CadeviationX2].Status.Homed AND arrAxisCtrl[AxiseNo.AxisName.CadeviationX2].Status.NoMoving AND
			arrAxisCtrl[AxiseNo.AxisName.CadeviationY].Status.Homed AND arrAxisCtrl[AxiseNo.AxisName.CadeviationY].Status.NoMoving	 THEN
			arrAxisCtrl[AxiseNo.AxisName.CaCarryingLine2].Cmd.bHome:=FALSE;//负极搬运平移2
			arrAxisCtrl[AxiseNo.AxisName.CaDTCarryingLine].Cmd.bHome:=FALSE;//负极叠片搬运平移		
			arrAxisCtrl[AxiseNo.AxisName.CadeviationX1].Cmd.bHome:=FALSE;//负极纠偏X1	
			arrAxisCtrl[AxiseNo.AxisName.CadeviationX2].Cmd.bHome:=FALSE;//负极纠偏X2
			arrAxisCtrl[AxiseNo.AxisName.CadeviationY].Cmd.bHome:=FALSE;//负极纠偏Y
			Ca_Carrying2TorMark:=FALSE;//负极搬运2平移力矩判断标志位
			Ca_GohomeTon.IN:=FALSE;
			Step_InitCaDT:=80;
		ELSIF arrAxisCtrl[AxiseNo.AxisName.CaCarryingLine2].Status.Error OR arrAxisCtrl[AxiseNo.AxisName.CadeviationX1].Status.Error OR 
				 arrAxisCtrl[AxiseNo.AxisName.CadeviationX2].Status.Error OR arrAxisCtrl[AxiseNo.AxisName.CadeviationY].Status.Error THEN
				 arrAxisCtrl[AxiseNo.AxisName.CaCarryingLine2].Cmd.bHome:=FALSE;//负极搬运平移2
				arrAxisCtrl[AxiseNo.AxisName.CaDTCarryingLine].Cmd.bHome:=FALSE;//负极叠片搬运平移		
				arrAxisCtrl[AxiseNo.AxisName.CadeviationX1].Cmd.bHome:=FALSE;//负极纠偏X1	
				arrAxisCtrl[AxiseNo.AxisName.CadeviationX2].Cmd.bHome:=FALSE;//负极纠偏X2
				arrAxisCtrl[AxiseNo.AxisName.CadeviationY].Cmd.bHome:=FALSE;//负极纠偏Y
				Ca_GohomeTon.IN:=FALSE;
				Ca_Gohoming:=FALSE;//负极取片回原点中	
				Step_InitCaDT:=9999;
		END_IF
	END_IF
80://
	//负极送片搬运平移2
	IF arrAxisCtrl[AxiseNo.AxisName.CaCarryingLine2].Status.Homed AND arrAxisCtrl[AxiseNo.AxisName.CaCarryingLine2].Status.NoMoving THEN
		IF arrAxisCtrl[AxiseNo.AxisName.CaCarryingLine2].Cmd.arrbRealPoint[1]  THEN
			arrAxisCtrl[AxiseNo.AxisName.CaCarryingLine2].Cmd.iGoSetPos:=0;
		ELSE
		   arrAxisCtrl[AxiseNo.AxisName.CaCarryingLine2].Cmd.iGoSetPos:=1;
		END_IF
	END_IF		
	//负极纠偏X1初始位
	IF arrAxisCtrl[AxiseNo.AxisName.CadeviationX1].Status.Homed AND arrAxisCtrl[AxiseNo.AxisName.CadeviationX1].Status.NoMoving THEN
		IF arrAxisCtrl[AxiseNo.AxisName.CadeviationX1].Cmd.arrbRealPoint[1]   THEN
			arrAxisCtrl[AxiseNo.AxisName.CadeviationX1].Cmd.iGoSetPos:=0;
		ELSE
		   arrAxisCtrl[AxiseNo.AxisName.CadeviationX1].Cmd.iGoSetPos:=1;
		END_IF	
	END_IF	
	//负极纠偏X2初始位
	IF arrAxisCtrl[AxiseNo.AxisName.CadeviationX2].Status.Homed AND arrAxisCtrl[AxiseNo.AxisName.CadeviationX2].Status.NoMoving THEN
		IF arrAxisCtrl[AxiseNo.AxisName.CadeviationX2].Cmd.arrbRealPoint[1]   THEN
			arrAxisCtrl[AxiseNo.AxisName.CadeviationX2].Cmd.iGoSetPos:=0;
		ELSE
		   arrAxisCtrl[AxiseNo.AxisName.CadeviationX2].Cmd.iGoSetPos:=1;
		END_IF	
	END_IF	
	//负极纠偏Y初始位
	IF arrAxisCtrl[AxiseNo.AxisName.CadeviationY].Status.Homed AND arrAxisCtrl[AxiseNo.AxisName.CadeviationY].Status.NoMoving THEN
		IF arrAxisCtrl[AxiseNo.AxisName.CadeviationY].Cmd.arrbRealPoint[1]   THEN
			arrAxisCtrl[AxiseNo.AxisName.CadeviationY].Cmd.iGoSetPos:=0;
		ELSE
		   arrAxisCtrl[AxiseNo.AxisName.CadeviationY].Cmd.iGoSetPos:=1;
		END_IF	
	END_IF		
	IF arrAxisCtrl[AxiseNo.AxisName.CaCarryingLine2].Cmd.arrbRealPoint[1] AND arrAxisCtrl[AxiseNo.AxisName.CaCarryingLine2].Status.NoMoving AND  
		arrAxisCtrl[AxiseNo.AxisName.CadeviationX1].Cmd.arrbRealPoint[1]  AND arrAxisCtrl[AxiseNo.AxisName.CadeviationX1].Status.NoMoving AND
		arrAxisCtrl[AxiseNo.AxisName.CadeviationX2].Cmd.arrbRealPoint[1]  AND arrAxisCtrl[AxiseNo.AxisName.CadeviationX2].Status.NoMoving AND
		arrAxisCtrl[AxiseNo.AxisName.CadeviationY].Cmd.arrbRealPoint[1] AND arrAxisCtrl[AxiseNo.AxisName.CadeviationY].Status.NoMoving  THEN	
		Step_InitCaDT:=90;
	ELSIF arrAxisCtrl[AxiseNo.AxisName.CaCarryingLine2].Status.Error OR arrAxisCtrl[AxiseNo.AxisName.CadeviationX1].Status.Error OR
		arrAxisCtrl[AxiseNo.AxisName.CadeviationX2].Status.Error OR arrAxisCtrl[AxiseNo.AxisName.CadeviationY].Status.Error THEN
		Ca_Gohoming:=FALSE;//负极取片回原点中	
		Step_InitCaDT:=9999;
	END_IF
		
90://叠片平移搬运轴回原点
		 IF NOT Ca_GohomeTon.Q THEN
			IF   arrAxisCtrl[AxiseNo.AxisName.CaCarryingLine2].Cmd.arrbRealPoint[1]  THEN
					arrAxisCtrl[AxiseNo.AxisName.CaDTCarryingLine].Cmd.bHome:=TRUE;//负极叠片搬运平移
					Ca_DTCarryingTorMark:=TRUE;//负极叠台搬运平移力矩判断标志位
			END_IF
			Ca_GohomeTon.IN:=TRUE;	
		 ELSE
			Ca_GohomeTon.IN:=FALSE;	
			Step_InitCaDT:=100;
		 END_IF
100://判断叠片平移回原点是否完成
		IF NOT Ca_GohomeTon.Q THEN
			Ca_GohomeTon.IN:=TRUE;
		ELSE	
			IF arrAxisCtrl[AxiseNo.AxisName.CaDTCarryingLine].Status.Homed AND arrAxisCtrl[AxiseNo.AxisName.CaDTCarryingLine].Status.NoMoving THEN
				arrAxisCtrl[AxiseNo.AxisName.CaDTCarryingLine].Cmd.bHome:=FALSE;//负极叠片搬运平移
				Ca_DTCarryingTorMark:=FALSE;//负极叠台搬运平移力矩判断标志位
				Ca_GohomeTon.IN:=FALSE;
				Step_InitCaDT:=110;
			ELSIF arrAxisCtrl[AxiseNo.AxisName.CaDTCarryingLine].Status.Error THEN
				arrAxisCtrl[AxiseNo.AxisName.CaDTCarryingLine].Cmd.bHome:=FALSE;//负极叠片搬运平移
				Ca_GohomeTon.IN:=FALSE;
				Ca_Gohoming:=FALSE;//负极取片回原点中	
				Step_InitCaDT:=9999;												
			END_IF
		END_IF
110://轴移动至初始位
	//负极叠台搬运平移
	IF arrAxisCtrl[AxiseNo.AxisName.CaDTCarryingLine].Status.Homed AND arrAxisCtrl[AxiseNo.AxisName.CaDTCarryingLine].Status.NoMoving THEN
		IF arrAxisCtrl[AxiseNo.AxisName.CaDTCarryingLine].Cmd.arrbRealPoint[1]   THEN
			arrAxisCtrl[AxiseNo.AxisName.CaDTCarryingLine].Cmd.iGoSetPos:=0;
			Step_InitCaDT:=120;
		ELSIF arrAxisCtrl[AxiseNo.AxisName.CaDTCarryingLine].Status.Error THEN
				Ca_Gohoming:=FALSE;//负极取片回原点中	
				Step_InitCaDT:=9999;
		ELSE
		   	arrAxisCtrl[AxiseNo.AxisName.CaDTCarryingLine].Cmd.iGoSetPos:=1;
		END_IF	
	END_IF	
120:
	arrCyCtrl[arrCyNo.ElectValveName.CaCarryingVacuum1]	.Cmd.bOFF:=TRUE;//负极搬运1真空关
	arrCyCtrl[arrCyNo.ElectValveName.CaCarryingVacuum1]	.Cmd.bON:=FALSE;//负极搬运1真空关
	arrCyCtrl[arrCyNo.ElectValveName.CaCarryingVacuum2]	.Cmd.bOFF:=TRUE;//负极搬运2真空关
	arrCyCtrl[arrCyNo.ElectValveName.CaCarryingVacuumBark1]	.Cmd.bOFF:=TRUE;//负极搬运1破真空关
	arrCyCtrl[arrCyNo.ElectValveName.CaCarryingVacuumBark2]	.Cmd.bOFF:=TRUE;//负极搬运2破真空关
	arrCyCtrl[arrCyNo.ElectValveName.CadeviationVacuum]	.Cmd.bOFF:=TRUE;//负极纠偏平台真空关
	arrCyCtrl[arrCyNo.ElectValveName.CadeviationVacuumBark]	.Cmd.bOFF:=TRUE;//负极纠偏平台破真空关
	arrCyCtrl[arrCyNo.ElectValveName.CaDTCarryingVacuum]	.Cmd.bOFF:=TRUE;//负极叠FALSE片真空关
	arrCyCtrl[arrCyNo.ElectValveName.CaDTCarryingVacuumBark]	.Cmd.bOFF:=TRUE;//负极叠片搬运升降破真空关					
	//负极送片搬运升降2
	IF arrAxisCtrl[AxiseNo.AxisName.CaCarryingUpDown2].Status.Homed AND arrAxisCtrl[AxiseNo.AxisName.CaCarryingUpDown2].Status.NoMoving THEN
		IF arrAxisCtrl[AxiseNo.AxisName.CaCarryingUpDown2].Cmd.arrbRealPoint[4] THEN
			arrAxisCtrl[AxiseNo.AxisName.CaCarryingUpDown2].Cmd.iGoSetPos:=0;
		ELSE
			arrAxisCtrl[AxiseNo.AxisName.CaCarryingUpDown2].Cmd.iGoSetPos:=4;
		END_IF	
	END_IF
	//负极叠片搬运升降
	IF arrAxisCtrl[AxiseNo.AxisName.CaDTCarryingUpDown].Status.Homed AND arrAxisCtrl[AxiseNo.AxisName.CaDTCarryingUpDown].Status.NoMoving THEN
		IF arrAxisCtrl[AxiseNo.AxisName.CaDTCarryingUpDown].Cmd.arrbRealPoint[4]  THEN
			arrAxisCtrl[AxiseNo.AxisName.CaDTCarryingUpDown].Cmd.iGoSetPos:=0;
		ELSE
		   arrAxisCtrl[AxiseNo.AxisName.CaDTCarryingUpDown].Cmd.iGoSetPos:=4;
		END_IF	
	END_IF		
	IF arrAxisCtrl[AxiseNo.AxisName.CaCarryingUpDown2].Cmd.arrbRealPoint[4] AND arrAxisCtrl[AxiseNo.AxisName.CaCarryingUpDown2].Status.NoMoving  AND
		arrAxisCtrl[AxiseNo.AxisName.CaDTCarryingUpDown].Cmd.arrbRealPoint[4] AND arrAxisCtrl[AxiseNo.AxisName.CaDTCarryingUpDown].Status.NoMoving THEN
		Ca_GohomeDone:=TRUE;//负极取片回原点完成
		Ca_Gohoming:=FALSE;//负极取片回原点中	
		Step_InitCaDT:=0;
	ELSIF arrAxisCtrl[AxiseNo.AxisName.CaCarryingUpDown2].Status.Error OR arrAxisCtrl[AxiseNo.AxisName.CaDTCarryingUpDown].Status.Error THEN
		Ca_Gohoming:=FALSE;//负极取片回原点中	
		Step_InitCaDT:=9999;
	END_IF		
END_CASE
//负极皮带初始化
IF rCa_BeltGohome_TRIG.Q THEN
	Ca_BeltGohomeDone:=FALSE;
	Ca_BeltGohoming:=FALSE;
	Mach_Control.Ca_b.Ca_SegbeltFalg:=FALSE;
	Step_InitCaDT0:=0;
END_IF

//回原点超时报警	

	IF  Ca_BeltGohoming THEN
		IF NOT Ca_BeltGohomeOverTon.Q THEN
			    Ca_BeltGohomeOverTon.IN:=TRUE;
		ELSE
			IF Ca_BeltGohomeOverTon.Q THEN
			      Mach_Control.Ca_b.Error[20]:=TRUE;//负极皮带回原点超时报警	
			     Ca_BeltGohomeOverTon.IN:=FALSE;
			END_IF	 	 
		END_IF

	ELSE
		Ca_BeltGohomeOverTon.IN:=FALSE;
	END_IF



CASE Step_InitCaDT0 OF 
0://
	IF fCa_BeltGohome_TRIG.Q THEN
		Ca_StandbyStep2:=0;
		Ca_StandbyStep4:=0;
		//Par.stDT_date.Ca_betlCount.5 :=FALSE;
		//Par.stDT_date.Ca_betlCount.4 :=FALSE;
		//Par.stDT_date.Ca_betlCount.3 :=FALSE;
		//Par.stDT_date.Ca_betlCount.2 :=FALSE;
		//Par.stDT_date.Ca_betlCount.1 :=FALSE;
		//Par.stDT_date.Ca_betlCount.0:=FALSE;
		Ca_BeltGohoming:=TRUE;
		Step_InitCaDT0:=20;
	END_IF
20:
	Ca_BeltGohomeDone:=FALSE;
	Ca_BeltGohomeTon.IN:=FALSE;
	IF NOT Ca_BeltGohomeDone THEN
		Step_InitCaDT0:=30;
	END_IF
30:
	IF NOT Ca_BeltGohomeTon.Q THEN
		Ca_BeltGohomeTon.IN:=TRUE;
		arrAxisCtrl[AxiseNo.AxisName.CaCarryingUpDown1].Cmd.bHome:=TRUE;//
	ELSE
		IF arrAxisCtrl[AxiseNo.AxisName.CaCarryingUpDown1].Status.Homed AND arrAxisCtrl[AxiseNo.AxisName.CaCarryingUpDown1].Status.NoMoving THEN
			Ca_BeltGohomeTon.IN:=FALSE;	
			arrAxisCtrl[AxiseNo.AxisName.CaCarryingUpDown1].Cmd.bHome:=FALSE;//
			Step_InitCaDT0:=40;
		ELSIF arrAxisCtrl[AxiseNo.AxisName.CaCarryingUpDown1].Status.Error THEN
			Ca_BeltGohomeTon.IN:=FALSE;	
			arrAxisCtrl[AxiseNo.AxisName.CaCarryingUpDown1].Cmd.bHome:=FALSE;//
			Ca_BeltGohoming:=FALSE;
			Step_InitCaDT0:=9999;											
		END_IF								
	END_IF
40://
		IF NOT Ca_BeltGohomeTon.Q THEN
			Ca_BeltGohomeTon.IN:=TRUE;
			arrAxisCtrl[AxiseNo.AxisName.CaCarryingWhirling1].Cmd.bHome:=TRUE;//
			arrAxisCtrl[AxiseNo.AxisName.CaCarryingLine1].Cmd.bHome:=TRUE;//
			Ca_Carrying1TorMark:=TRUE;//负极搬运1平移力矩判断标志位
		ELSE
			IF arrAxisCtrl[AxiseNo.AxisName.CaCarryingWhirling1].Status.Homed AND arrAxisCtrl[AxiseNo.AxisName.CaCarryingWhirling1].Status.NoMoving AND 
				 arrAxisCtrl[AxiseNo.AxisName.CaCarryingLine1].Status.Homed AND arrAxisCtrl[AxiseNo.AxisName.CaCarryingLine1].Status.NoMoving THEN
				Ca_BeltGohomeTon.IN:=FALSE;	
				arrAxisCtrl[AxiseNo.AxisName.CaCarryingWhirling1].Cmd.bHome:=FALSE;//
				arrAxisCtrl[AxiseNo.AxisName.CaCarryingLine1].Cmd.bHome:=FALSE;//
				Ca_Carrying1TorMark:=FALSE;//负极搬运1平移力矩判断标志位
				Step_InitCaDT0:=50;
			ELSIF arrAxisCtrl[AxiseNo.AxisName.CaCarryingWhirling1].Status.Error OR arrAxisCtrl[AxiseNo.AxisName.CaCarryingLine1].Status.Error THEN
				Ca_BeltGohomeTon.IN:=FALSE;	
				arrAxisCtrl[AxiseNo.AxisName.CaCarryingWhirling1].Cmd.bHome:=FALSE;//
				arrAxisCtrl[AxiseNo.AxisName.CaCarryingLine1].Cmd.bHome:=FALSE;//
				Ca_BeltGohoming:=FALSE;
				Step_InitCaDT0:=9999;
			END_IF								
		END_IF	
50:
	IF arrAxisCtrl[AxiseNo.AxisName.CaCarryingWhirling1].Status.Homed AND arrAxisCtrl[AxiseNo.AxisName.CaCarryingWhirling1].Status.NoMoving THEN
		IF arrAxisCtrl[AxiseNo.AxisName.CaCarryingWhirling1].Cmd.arrbRealPoint[1]   THEN
			arrAxisCtrl[AxiseNo.AxisName.CaCarryingWhirling1].Cmd.iGoSetPos:=0;
		ELSE
		   arrAxisCtrl[AxiseNo.AxisName.CaCarryingWhirling1].Cmd.iGoSetPos:=1;
		END_IF	
	END_IF		

	IF arrAxisCtrl[AxiseNo.AxisName.CaCarryingUpDown1].Status.Homed AND arrAxisCtrl[AxiseNo.AxisName.CaCarryingUpDown1].Status.NoMoving THEN
		IF arrAxisCtrl[AxiseNo.AxisName.CaCarryingUpDown1].Cmd.arrbRealPoint[1]   THEN
			arrAxisCtrl[AxiseNo.AxisName.CaCarryingUpDown1].Cmd.iGoSetPos:=0;
		ELSE
		   arrAxisCtrl[AxiseNo.AxisName.CaCarryingUpDown1].Cmd.iGoSetPos:=1;
		END_IF	
	END_IF		

	IF arrAxisCtrl[AxiseNo.AxisName.CaCarryingLine1].Status.Homed AND arrAxisCtrl[AxiseNo.AxisName.CaCarryingLine1].Status.NoMoving THEN
		IF arrAxisCtrl[AxiseNo.AxisName.CaCarryingLine1].Cmd.arrbRealPoint[1]   THEN
			arrAxisCtrl[AxiseNo.AxisName.CaCarryingLine1].Cmd.iGoSetPos:=0;
		ELSE
		   arrAxisCtrl[AxiseNo.AxisName.CaCarryingLine1].Cmd.iGoSetPos:=1;
		END_IF	
	END_IF	

	IF 	arrAxisCtrl[AxiseNo.AxisName.CaCarryingLine1].Cmd.arrbRealPoint[1] AND	arrAxisCtrl[AxiseNo.AxisName.CaCarryingWhirling1].Cmd.arrbRealPoint[1]  AND 
		 arrAxisCtrl[AxiseNo.AxisName.CaCarryingWhirling1].Cmd.arrbRealPoint[1] THEN
		 Ca_BeltGohomeDone:=TRUE;
		 Ca_BeltGohoming:=FALSE;
		 Step_InitCaDT0:=0;
	ELSIF  arrAxisCtrl[AxiseNo.AxisName.CaCarryingLine1].Status.Error OR arrAxisCtrl[AxiseNo.AxisName.CaCarryingWhirling1].Status.Error THEN
		Ca_BeltGohoming:=FALSE;
		Step_InitCaDT0:=9999;
	END_IF
						
END_CASE

END_IF
END_ACTION

ACTION Ca_OverNG:


(*******************************************************************************************************踢f负极对齐度NG片**************************************************************************************************************************)
 IF   Ca_OverNGStep=1630 THEN
	arrAxisCtrl[AxiseNo.AxisName.CaDTCarryingUpDown].Cmd.fOverride:=50;
 ELSE
   arrAxisCtrl[AxiseNo.AxisName.CaDTCarryingUpDown].Cmd.fOverride:=100;
 END_IF


IF Mach_Control.U.DT_iMode=1 THEN//在自动状态下
   CASE Ca_OverNGStep OF   
			1000://判断负极叠台搬运是否有片，有片的话放到纠偏台
						fAnScaling:=1;//20240508 CF
			            fCaScaling:=1;//20240508 CF		
						CaOverNGcount:=CaOverNGcount+1;
						IF arrCyCtrl[arrCyNo.ElectValveName.CaDTCarryingVacuum].Io.DIOnSwitch AND  Mach_Control.Ca_b.Ca_DPCarryingFalg  THEN//负极再取片位且叠台搬运有片,把当前片放到纠偏台
							Ca_OverNGStep:=1010;
						ELSE
							Ca_OverNGStep:=1050;	
						END_IF
	
			1010://纠偏台回初始位
				//纠偏平台X1移动至初始位
				IF NOT DP_SinStepe THEN
					IF arrAxisCtrl[AxiseNo.AxisName.CadeviationX1].Status.Homed  AND arrAxisCtrl[AxiseNo.AxisName.CadeviationX1].Status.NoMoving AND NOT  arrAxisCtrl[AxiseNo.AxisName.CadeviationX1].Status.Error THEN
						IF arrAxisCtrl[AxiseNo.AxisName.CadeviationX1].Cmd.arrbRealPoint[1] THEN
							arrAxisCtrl[AxiseNo.AxisName.CadeviationX1].Cmd.iGoSetPos:=0;
						ELSE
							arrAxisCtrl[AxiseNo.AxisName.CadeviationX1].Cmd.iGoSetPos:=1;
						END_IF					
					END_IF
					//纠偏平台X2移动至初始位
					IF arrAxisCtrl[AxiseNo.AxisName.CadeviationX2].Status.Homed  AND arrAxisCtrl[AxiseNo.AxisName.CadeviationX2].Status.NoMoving AND NOT  arrAxisCtrl[AxiseNo.AxisName.CadeviationX2].Status.Error THEN
						IF arrAxisCtrl[AxiseNo.AxisName.CadeviationX2].Cmd.arrbRealPoint[1] THEN
							arrAxisCtrl[AxiseNo.AxisName.CadeviationX2].Cmd.iGoSetPos:=0;
						ELSE
							arrAxisCtrl[AxiseNo.AxisName.CadeviationX2].Cmd.iGoSetPos:=1;
						END_IF					
					END_IF
					//纠偏平台X2移动至初始位
					IF arrAxisCtrl[AxiseNo.AxisName.CadeviationY].Status.Homed  AND arrAxisCtrl[AxiseNo.AxisName.CadeviationY].Status.NoMoving AND NOT  arrAxisCtrl[AxiseNo.AxisName.CadeviationY].Status.Error THEN
						IF arrAxisCtrl[AxiseNo.AxisName.CadeviationY].Cmd.arrbRealPoint[1] THEN
							arrAxisCtrl[AxiseNo.AxisName.CadeviationY].Cmd.iGoSetPos:=0;
						ELSE
							arrAxisCtrl[AxiseNo.AxisName.CadeviationY].Cmd.iGoSetPos:=1;
						END_IF					
					END_IF
					IF arrAxisCtrl[AxiseNo.AxisName.CadeviationX1].Cmd.arrbRealPoint[1] AND arrAxisCtrl[AxiseNo.AxisName.CadeviationX2].Cmd.arrbRealPoint[1] AND arrAxisCtrl[AxiseNo.AxisName.CadeviationY].Cmd.arrbRealPoint[1] THEN
						DT_SingeMode();//单步选择	
						Ca_OverNGStep:=1020;
                        DT_TON[4].IN:=FALSE;	
					END_IF	
				END_IF
			1020://叠台搬运极片放回纠偏台
				IF NOT DP_SinStepe THEN
					IF arrAxisCtrl[AxiseNo.AxisName.CaDTCarryingLine].Cmd.arrbRealPoint[1]  AND NOT Mach_Control.Ca_b.Ca_deviationFalg THEN 
						IF arrAxisCtrl[AxiseNo.AxisName.CaDTCarryingUpDown].Cmd.arrbRealPoint[2] THEN
							arrAxisCtrl[AxiseNo.AxisName.CaDTCarryingUpDown].Cmd.iGoSetPos:=0;
					    ELSE
							arrAxisCtrl[AxiseNo.AxisName.CaDTCarryingUpDown].Cmd.iGoSetPos:=2;//负极d叠台搬运下降至取片位
					    END_IF
                   END_IF
				       IF arrAxisCtrl[AxiseNo.AxisName.CaDTCarryingUpDown].Cmd.arrbRealPoint[2] THEN
				           	/// 吸盘破真空    纠偏台开真空
							arrCyCtrl[arrCyNo.ElectValveName.CaDTCarryingVacuum].Cmd.bON:=TRUE;	//负极叠台搬运升降真空	真空
							arrCyCtrl[arrCyNo.ElectValveName.CaDTCarryingVacuum].Cmd.bOFF:=FALSE;	//负极叠台搬运升降真空破真空								
							arrCyCtrl[arrCyNo.ElectValveName.CadeviationVacuum].Cmd.bON:=TRUE;	//负极纠偏台真空			
							arrCyCtrl[arrCyNo.ElectValveName.CadeviationVacuum].Cmd.bOFF:=FALSE;	//负极纠偏台真空	   
							DT_SingeMode();//单步选择	
							Ca_OverNGStep:=1030;
							DT_TON[4].IN:=TRUE;
							Mach_Control.Ca_b.Ca_deviationFalg:=TRUE;//置位位纠偏平台有料标记
							Mach_Control.Ca_b.Ca_DPCarryingFalg:=FALSE;//负极搬运真空吸盘有料标记复位							
	                    END_IF
				END_IF
			1030://叠台搬运极片上升至凸轮耦合初始高度
				IF NOT DP_SinStepe AND DT_TON[4].Q THEN
					IF arrAxisCtrl[AxiseNo.AxisName.CaDTCarryingUpDown].Cmd.arrbRealPoint[4] THEN
						arrAxisCtrl[AxiseNo.AxisName.CaDTCarryingUpDown].Cmd.iGoSetPos:=0;
						/// 吸盘破真空    纠偏台开真空
						Mach_Control.Ca_b.Ca_deviationFalg:=TRUE;//置位位纠偏平台有料标记
						Mach_Control.Ca_b.Ca_DPCarryingFalg:=FALSE;//负极搬运真空吸盘有料标记复位
						Par.stDT_date.Ca_MQ_Slice[8]:=Par.stDT_date.Ca_MQ_Slice[9];
						DT_SingeMode();//单步选择	
						Ca_OverNGStep:=1050;
						DT_TON[4].IN:=FALSE;
					ELSE
						arrAxisCtrl[AxiseNo.AxisName.CaDTCarryingUpDown].Cmd.iGoSetPos:=4;//负极搬运升降2上升至凸轮耦合初始高度
					END_IF			
				END_IF		   
		
            1050://判断主轴是否停止、是否在初始位、是否有轴在耦合中
					IF NOT DP_SinStepe THEN
								IF arrAxis[AxiseNo.VirAxisName.VirMain].Status.NotMoving AND arrAxis[AxiseNo.VirAxisName.VirMain].NcToPlc.SetPos=0 AND NOT DT_AxiseCoupling THEN
									DT_SingeMode();//单步选择
									Ca_OverNGStep:=1070;
								ELSE
									DP_Step1:=100;//调用主轴回初始位子程序
									DT_SingeMode();//单步选择
									Ca_OverNGStep:=1060;
								END_IF
			    	END_IF		
			1060://判断主轴的模长的当前位置是否为0
				IF NOT DP_SinStepe THEN
					IF DP_Step1=6666 AND arrAxis[AxiseNo.VirAxisName.VirMain].Status.NotMoving AND arrAxis[AxiseNo.VirAxisName.VirMain].NcToPlc.SetPos=0 AND NOT DT_AxiseCoupling  THEN
						DT_SingeMode();//单步选择
						Ca_OverNGStep:=1070;
					END_IF	
				END_IF							

